// TIA Portal V20 export
DATA_BLOCK "InstCallEquipment"   // DB119
{ DB_Accessible_From_OPC_UA := 'FALSE' }
AUTHOR : ERsystem_FA2_DH. Kim
// stored: AssignedProDiagFB Unit1.Em5.ProDiag, DBAccessibleFromOPCUA false, DBAccessibleFromWebserver false, InstanceOfName Unit1.Em5.CallEquipment, InstanceOfType FB, Namespace Unit1.Em5
"Unit1.Em5.CallEquipment"
   // VAR_INPUT
   //    ZoneOperationEnable { ExternalWritable := 'False'} : "LWONIK_typeSafetyZoneManualOperation";
   // END_VAR
   // VAR_IN_OUT
   //    unitStatus : "LAF_typeUnitStatus";
   //    unitAlarmDB : "LAF_typeAlarms";
   //    emFeedback : "LUC_typeEmFeedback";
   // END_VAR
   // VAR
   //    InstSequenceMainPnP { S7_SetPoint := 'True'} : "Unit1.Em5.Sequence_1_MainPnP";
   //    InstSequenceAlignTable { S7_SetPoint := 'True'} : "Unit1.Em5.Sequence_2_AlignTable";
   //    InstSequenceNgPnP { S7_SetPoint := 'True'} : "Unit1.Em5.Sequence_3_NgPnP";
   //    InstSequenceGaugeRnR : "Unit1.Em5.Sequence_10_GaugeRnR";
   //    instMainPnPHomeJob10 : "LAF_SelectJob";
   //    instMainPnPHomeJob1 : "LAF_SelectJob";
   //    instMainPnPLoadJob2 : "LAF_SelectJob";
   //    instMainPnPUnloadJob3 : "LAF_SelectJob";
   //    instMainPnPAvoidJob4 : "LAF_SelectJob";
   //    instMainPnPOneLoadJob5 : "LAF_SelectJob";
   //    instMainPnPOneUnLoadJob6 : "LAF_SelectJob";
   //    instAlignTableHomeJob1 : "LAF_SelectJob";
   //    instAlignTableLoadJob2 : "LAF_SelectJob";
   //    instAlignTableVisionJob3 : "LAF_SelectJob";
   //    instAlignTableUnloadJob4 : "LAF_SelectJob";
   //    instAlignTableMotionJob22 : "LAF_SelectJob";
   //    instNgPnPHomeJob1 : "LAF_SelectJob";
   //    instNgPnPLoadJob2 : "LAF_SelectJob";
   //    instNgPnPUnloadJob3 : "LAF_SelectJob";
   //    instGaugeRnRCommonReadyJob1 : "LAF_SelectJob";
   //    instGaugeRnRCommonGetMasterPieceJob2 : "LAF_SelectJob";
   //    instGaugeRnRCommonMainPnPMoveAlignTableStackTableJob3 : "LAF_SelectJob";
   //    instGaugeRnRCommonMainPnp1ToAlignTableJob4 : "LAF_SelectJob";
   //    instGaugeRnRCommonMainPnPMoveReelCutConvyorAlignTableJob5 : "LAF_SelectJob";
   //    instGaugeRnRCommonAlignTableVisionAdjustJob6 : "LAF_SelectJob";
   //    instGaugeRnR1AlignAlignTableToMainPnP1Job10 { S7_SetPoint := 'True'} : "LAF_SelectJob";
   //    instGaugeRnR1AlignMainPnPMoveReelCutConvyorAlignTableJob11 { S7_SetPoint := 'True'} : "LAF_SelectJob";
   //    instGaugeRnR1AlignAlignTableMoveWaitJob12 { S7_SetPoint := 'True'} : "LAF_SelectJob";
   //    instGaugeRnR1AlignUnloadMasterPieceJob13 { S7_SetPoint := 'True'} : "LAF_SelectJob";
   //    instGaugeRnR1StackMainPnPMoveReelCutConvyorAlignTableJob15 { S7_SetPoint := 'True'} : "LAF_SelectJob";
   //    instGaugeRnR1StackAlignTableToMainPnP2Job16 { S7_SetPoint := 'True'} : "LAF_SelectJob";
   //    instGaugeRnR1StackMainPnPMoveAlignTableJob17 { S7_SetPoint := 'True'} : "LAF_SelectJob";
   //    instGaugeRnR1StackAlignTableMoveWaitJob18 { S7_SetPoint := 'True'} : "LAF_SelectJob";
   //    instGaugeRnR1StackMainPnP2ToStackTableJob19 { S7_SetPoint := 'True'} : "LAF_SelectJob";
   //    instGaugeRnR1StackStackTableToMainPnP2Job20 { S7_SetPoint := 'True'} : "LAF_SelectJob";
   //    instGaugeRnR1StackMainPnPMoveReelCutConvyorAlignTableJob21 { S7_SetPoint := 'True'} : "LAF_SelectJob";
   //    instGaugeRnR1StackMainPnP2ToAlignTableJob22 { S7_SetPoint := 'True'} : "LAF_SelectJob";
   //    instGaugeRnR1StackMainPnPMoveAlignTableJob23 { S7_SetPoint := 'True'} : "LAF_SelectJob";
   //    instGaugeRnR1StackAlignTableToMainPnP1Job24 { S7_SetPoint := 'True'} : "LAF_SelectJob";
   //    instGaugeRnR1StackMainPnPMoveReelCutConvyorAlignTableJob25 { S7_SetPoint := 'True'} : "LAF_SelectJob";
   //    instGaugeRnR1StackUnloadMasterPieceJob26 { S7_SetPoint := 'True'} : "LAF_SelectJob";
   //    instGaugeRnR3AlignMainPnPMoveReelCutConvyorAlignTableJob30 { S7_SetPoint := 'True'} : "LAF_SelectJob";
   //    instGaugeRnR3AlignNGPnPLoadMasterPieceJob31 { S7_SetPoint := 'True'} : "LAF_SelectJob";
   //    instGaugeRnR3AlignMainPnP2MoveAlignTableJob32 { S7_SetPoint := 'True'} : "LAF_SelectJob";
   //    instGaugeRnR3AlignAlignTableMoveWaitJob33 { S7_SetPoint := 'True'} : "LAF_SelectJob";
   //    instGaugeRnRCommonCheckCompleteJob39 { S7_SetPoint := 'True'} : "LAF_SelectJob";
   //    instCmPnp1stCathodeDetectSensor { S7_SetPoint := 'True'} : "LBC_DigitalSignalCn";
   //    instCmPnp2ndCathodeDetectSensor { S7_SetPoint := 'True'} : "LBC_DigitalSignalCn";
   //    instCmCathodeAlignTableElectrodeDetectSensor { S7_SetPoint := 'True'} : "LBC_DigitalSignalCn";
   //    instCmCathodeNgBoxFullSensorDetectSensor { S7_SetPoint := 'True'} : "LBC_DigitalSignalCn";
   //    instCmCathodeNgBoxDetectSensor { S7_SetPoint := 'True'} : "LBC_DigitalSignalCn";
   //    instCmCathodeMainPnP1AxisX { S7_SetPoint := 'True'} : "LBC_Axis64Pos_TecPlcCn";
   //    instCmCathodeMainPnP2AxisX { S7_SetPoint := 'True'} : "LBC_Axis64Pos_TecPlcCn";
   //    instCmCathodeMainPnP1AxisY { S7_SetPoint := 'True'} : "LBC_Axis64Pos_TecPlcCn";
   //    instCmCathodeMainPnP1AxisZ { S7_SetPoint := 'True'} : "LBC_Axis64Pos_TecPlcCn";
   //    instCmCathodeMainPnP2AxisZ { S7_SetPoint := 'True'} : "LBC_Axis64Pos_TecPlcCn";
   //    instCmCathodeAlignTableAxisX { S7_SetPoint := 'True'} : "LBC_Axis64Pos_TecPlcCn";
   //    instCmCathodeAlignTableAxisY1 { S7_SetPoint := 'True'} : "LBC_Axis64Pos_TecPlcCn";
   //    instCmCathodeAlignTableAxisY2 { S7_SetPoint := 'True'} : "LBC_Axis64Pos_TecPlcCn";
   //    instInterlockCathodeMainPnP1AxisX { S7_SetPoint := 'True'} : "LER_Axis64Pos_InterlockSummary";
   //    instInterlockCathodeMainPnP1AxisY { S7_SetPoint := 'True'} : "LER_Axis64Pos_InterlockSummary";
   //    instInterlockCathodeMainPnP1AxisZ { S7_SetPoint := 'True'} : "LER_Axis64Pos_InterlockSummary";
   //    instInterlockCathodeMainPnP2AxisX { S7_SetPoint := 'True'} : "LER_Axis64Pos_InterlockSummary";
   //    instInterlockCathodeMainPnP2AxisZ { S7_SetPoint := 'True'} : "LER_Axis64Pos_InterlockSummary";
   //    instInterlockCathodeAlignTableAxisX { S7_SetPoint := 'True'} : "LER_Axis64Pos_InterlockSummary";
   //    instInterlockCathodeAlignTableAxisY1 { S7_SetPoint := 'True'} : "LER_Axis64Pos_InterlockSummary";
   //    instInterlockCathodeAlignTableAxisY2 { S7_SetPoint := 'True'} : "LER_Axis64Pos_InterlockSummary";
   //    instCathodeMainPnP1AxisXSoftCam : "LER_SoftCam_Interface";
   //    instCathodeMainPnP2AxisXSoftCam { S7_SetPoint := 'True'} : "LER_SoftCam_Interface";
   //    instCathodeMainPnP1AxisYSoftCam { S7_SetPoint := 'True'} : "LER_SoftCam_Interface";
   //    instCathodeMainPnP1AxisZSoftCam { S7_SetPoint := 'True'} : "LER_SoftCam_Interface";
   //    instCathodeMainPnP2AxisZSoftCam { S7_SetPoint := 'True'} : "LER_SoftCam_Interface";
   //    instCathodeAlignTableAxisXSoftCam { S7_SetPoint := 'True'} : "LER_SoftCam_Interface";
   //    instCathodeAlignTableAxisY1SoftCam { S7_SetPoint := 'True'} : "LER_SoftCam_Interface";
   //    instCathodeAlignTableAxisY2SoftCam { S7_SetPoint := 'True'} : "LER_SoftCam_Interface";
   //    instCmCathodeMainPnP1RotaryCwCcw { ExternalAccessible := 'False'; ExternalVisible := 'False'; ExternalWritable := 'False'} : "LBC_TwoWayActuatorCn";
   //    instCmCathodeMainPnP1stSuctionPlateVacuum { ExternalAccessible := 'False'; ExternalVisible := 'False'; ExternalWritable := 'False'} : "LBC_TwoWayActuatorCn";
   //    instCmCathodeMainPnP2ndSuctionPlateVacuum { ExternalAccessible := 'False'; ExternalVisible := 'False'; ExternalWritable := 'False'} : "LBC_TwoWayActuatorCn";
   //    instCmCathodeAlignTableSuctionPlateVacuum { ExternalAccessible := 'False'; ExternalVisible := 'False'; ExternalWritable := 'False'; S7_SetPoint := 'True'} : "LBC_TwoWayActuatorCn";
   //    instCmCathodeGlassCleaning { ExternalAccessible := 'False'; ExternalVisible := 'False'; ExternalWritable := 'False'; S7_SetPoint := 'True'} : "LBC_TwoWayActuatorCn";
   //    instCmCathodeNgPnpUpDown { ExternalAccessible := 'False'; ExternalVisible := 'False'; ExternalWritable := 'False'; S7_SetPoint := 'True'} : "LBC_TwoWayActuatorCn";
   //    instCmCathodeNgPnp1stFwdBwd { ExternalAccessible := 'False'; ExternalVisible := 'False'; ExternalWritable := 'False'; S7_SetPoint := 'True'} : "LBC_TwoWayActuatorCn";
   //    instCmCathodeNgPnp2ndFwdBwd { ExternalAccessible := 'False'; ExternalVisible := 'False'; ExternalWritable := 'False'; S7_SetPoint := 'True'} : "LBC_TwoWayActuatorCn";
   //    instCmCathodeMaintenanceMovingFixFwdBwd { ExternalAccessible := 'False'; ExternalVisible := 'False'; ExternalWritable := 'False'; S7_SetPoint := 'True'} : "LBC_TwoWayActuatorCn";
   //    instCmCathodeNgBoxLiftUpDown { ExternalAccessible := 'False'; ExternalVisible := 'False'; ExternalWritable := 'False'; S7_SetPoint := 'True'} : "LBC_TwoWayActuatorCn";
   //    instCmCathodeNgBoxLockUpDown { ExternalAccessible := 'False'; ExternalVisible := 'False'; ExternalWritable := 'False'; S7_SetPoint := 'True'} : "LBC_TwoWayActuatorCn";
   //    instCmCathodeNgPnpVaccum { ExternalAccessible := 'False'; ExternalVisible := 'False'; ExternalWritable := 'False'; S7_SetPoint := 'True'} : "LBC_TwoWayActuatorCn";
   //    instCmCathodeConveyorCoverFwdBwd { S7_SetPoint := 'True'} : "LBC_TwoWayActuatorCn";
   //    instCmCathodeConveyorPickUpBlower { S7_SetPoint := 'True'} : "LBC_TwoWayActuatorCn";
   //    instCmCathodeVisionControllerInterface { ExternalAccessible := 'False'; ExternalVisible := 'False'; ExternalWritable := 'False'; S7_SetPoint := 'True'} : "LER_Vision_XGX2000";
   //    instAlignVisionConversion : "LER_AlignVisionConversion";
   //    instManageAlarms { ExternalWritable := 'False'} : "LAF_ManageAlarms";
   //    instEventsPFE : "Unit1.Em5.EventsPFE";
   //    instLER_BrakeTestCathodeMainPnP1AxisZ : "LER_BrakeTest";
   //    instLER_BrakeTestCathodeMainPnP2AxisZ { S7_SetPoint := 'True'} : "LER_BrakeTest";
   //    statUnitStatus { ExternalWritable := 'False'} : "LAF_typeUnitStatus";
   //    statSlmStatus : Struct
   //       running { ExternalWritable := 'False'} : Bool;
   //       powerOff { ExternalWritable := 'False'} : Bool;
   //    END_STRUCT;
   //    statAllBrakeTest { ExternalWritable := 'False'} : "LER_typeBrakeTestUnitCommands";
   //    statTonTime { ExternalAccessible := 'False'; ExternalVisible := 'False'; ExternalWritable := 'False'} : Array[0..1999] of TON_TIME;
   //    statTofTime { ExternalAccessible := 'False'; ExternalVisible := 'False'; ExternalWritable := 'False'} : Array[0..99] of TOF_TIME;
   //    statPulse { ExternalAccessible := 'False'; ExternalVisible := 'False'; ExternalWritable := 'False'} : Struct
   //       miscellaneous : Array[0..99] of Bool;
   //       workingDone : Struct
   //          mainPnP : Array[0..99] of Bool;
   //          alignTable : Array[0..99] of Bool;
   //          ngPnP : Array[0..99] of Bool;
   //       END_STRUCT;
   //       axisEnable : Array[0..99] of Bool;
   //       brakeTest : Array[0..99] of Bool;
   //    END_STRUCT;
   //    statEnableManualCmds : Bool := TRUE;
   //    Scan_on : Bool;
   //    "*** Interlock Axis ***" { ExternalAccessible := 'False'; ExternalVisible := 'False'; ExternalWritable := 'False'} : Bool;
   //    "cathodeMainPnP1AxisX Home" { S7_SetPoint := 'True'} : "Homing.LER_Axis";
   //    "cathodeMainPnP1AxisX Jog_CW" { S7_SetPoint := 'True'} : "Jog.LER_Axis";
   //    "cathodeMainPnP1AxisX Jog_CCW" { S7_SetPoint := 'True'} : "Jog.LER_Axis";
   //    "cathodeMainPnP1AxisX Position_" { S7_SetPoint := 'True'} : Array[0..5] of "Position.LER_Axis";
   //    "cathodeMainPnP2AxisX Home" { S7_SetPoint := 'True'} : "Homing.LER_Axis";
   //    "cathodeMainPnP2AxisX Jog_CW" { S7_SetPoint := 'True'} : "Jog.LER_Axis";
   //    "cathodeMainPnP2AxisX Jog_CCW" { S7_SetPoint := 'True'} : "Jog.LER_Axis";
   //    "cathodeMainPnP2AxisX Position_" { S7_SetPoint := 'True'} : Array[0..5] of "Position.LER_Axis";
   //    "cathodeMainPnP1AxisY Home" { S7_SetPoint := 'True'} : "Homing.LER_Axis";
   //    "cathodeMainPnP1AxisY Jog_CW" { S7_SetPoint := 'True'} : "Jog.LER_Axis";
   //    "cathodeMainPnP1AxisY Jog_CCW" { S7_SetPoint := 'True'} : "Jog.LER_Axis";
   //    "cathodeMainPnP1AxisY Position_" { S7_SetPoint := 'True'} : Array[0..5] of "Position.LER_Axis";
   //    "cathodeMainPnP1AxisZ Home" { S7_SetPoint := 'True'} : "Homing.LER_Axis";
   //    "cathodeMainPnP1AxisZ Jog_CW" { S7_SetPoint := 'True'} : "Jog.LER_Axis";
   //    "cathodeMainPnP1AxisZ Jog_CCW" { S7_SetPoint := 'True'} : "Jog.LER_Axis";
   //    "cathodeMainPnP1AxisZ Position_" { S7_SetPoint := 'True'} : Array[0..5] of "Position.LER_Axis";
   //    "cathodeMainPnP2AxisZ Home" { S7_SetPoint := 'True'} : "Homing.LER_Axis";
   //    "cathodeMainPnP2AxisZ Jog_CW" { S7_SetPoint := 'True'} : "Jog.LER_Axis";
   //    "cathodeMainPnP2AxisZ Jog_CCW" { S7_SetPoint := 'True'} : "Jog.LER_Axis";
   //    "cathodeMainPnP2AxisZ Position_" { S7_SetPoint := 'True'} : Array[0..5] of "Position.LER_Axis";
   //    "cathodeAlignTableAxisX Home" { S7_SetPoint := 'True'} : "Homing.LER_Axis";
   //    "cathodeAlignTableAxisX Jog_CW" { S7_SetPoint := 'True'} : "Jog.LER_Axis";
   //    "cathodeAlignTableAxisX Jog_CCW" { S7_SetPoint := 'True'} : "Jog.LER_Axis";
   //    "cathodeAlignTableAxisX Position_" { S7_SetPoint := 'True'} : Array[0..5] of "Position.LER_Axis";
   //    "cathodeAlignTableAxisY1 Home" { S7_SetPoint := 'True'} : "Homing.LER_Axis";
   //    "cathodeAlignTableAxisY1 Jog_CW" { S7_SetPoint := 'True'} : "Jog.LER_Axis";
   //    "cathodeAlignTableAxisY1 Jog_CCW" { S7_SetPoint := 'True'} : "Jog.LER_Axis";
   //    "cathodeAlignTableAxisY1 Position_" { S7_SetPoint := 'True'} : Array[0..5] of "Position.LER_Axis";
   //    "cathodeAlignTableAxisY2 Home" { S7_SetPoint := 'True'} : "Homing.LER_Axis";
   //    "cathodeAlignTableAxisY2 Jog_CW" { S7_SetPoint := 'True'} : "Jog.LER_Axis";
   //    "cathodeAlignTableAxisY2 Jog_CCW" { S7_SetPoint := 'True'} : "Jog.LER_Axis";
   //    "cathodeAlignTableAxisY2 Position_" { S7_SetPoint := 'True'} : Array[0..5] of "Position.LER_Axis";
   //    "*** Interlock Actuator ******" { ExternalAccessible := 'False'; ExternalVisible := 'False'; ExternalWritable := 'False'} : Bool;
   //    "cathodeNgBoxLiftUpDown Home" { S7_SetPoint := 'True'} : "Cylinder.LER_Actuator";
   //    "cathodeNgBoxLiftUpDown Work" { S7_SetPoint := 'True'} : "Cylinder.LER_Actuator";
   //    "cathodeNgBoxLockUpDown Home" { S7_SetPoint := 'True'} : "Cylinder.LER_Actuator";
   //    "cathodeNgBoxLockUpDown Work" { S7_SetPoint := 'True'} : "Cylinder.LER_Actuator";
   //    "cathodeMaintenanceMovingFixFrontFwdBwd Home" { S7_SetPoint := 'True'} : "Cylinder.LER_Actuator";
   //    "cathodeMaintenanceMovingFixFrontFwdBwd Work" { S7_SetPoint := 'True'} : "Cylinder.LER_Actuator";
   //    "cathodeGlassCleaning Home" { S7_SetPoint := 'True'} : "Cylinder.LER_Actuator";
   //    "cathodeGlassCleaning Work" { S7_SetPoint := 'True'} : "Cylinder.LER_Actuator";
   //    "cathodeNgPnp1stFwdBwd Home" { S7_SetPoint := 'True'} : "Cylinder.LER_Actuator";
   //    "cathodeNgPnp1stFwdBwd Work" { S7_SetPoint := 'True'} : "Cylinder.LER_Actuator";
   //    "cathodeNgPnpUpDown Home" { S7_SetPoint := 'True'} : "Cylinder.LER_Actuator";
   //    "cathodeNgPnpUpDown Work" { S7_SetPoint := 'True'} : "Cylinder.LER_Actuator";
   //    "cathodeMainPnP1RotaryCwCcw Home" { S7_SetPoint := 'True'} : "Cylinder.LER_Actuator";
   //    "cathodeMainPnP1RotaryCwCcw Work" { S7_SetPoint := 'True'} : "Cylinder.LER_Actuator";
   //    "cathodeNgPnp2ndFwdBwd Home" { S7_SetPoint := 'True'} : "Cylinder.LER_Actuator";
   //    "cathodeNgPnp2ndFwdBwd Work" { S7_SetPoint := 'True'} : "Cylinder.LER_Actuator";
   //    Tracking_05 { S7_SetPoint := 'True'} : "Unit1.Em5.PartData";
   //    AXIS7 : "LER_CM_Name";
   //    AXIS13 : "LER_CM_Name";
   //    AXIS18 : "LER_CM_Name";
   //    Cylinder23 : "LER_CM_Name";
   //    Cylinder28 : "LER_CM_Name";
   //    Vaccum15 : "LER_CM_Name";
   //    instAlignVisionHistory { S7_SetPoint := 'True'} : "LER_visionHistory";
   //    instAlignCalibration { S7_SetPoint := 'True'} : "LER_AlignCalibration";
   //    instAlignMoveCalibration { S7_SetPoint := 'True'} : "LER_AlignMoveCalibration";
   //    instAlignThetaCalibration { S7_SetPoint := 'True'} : "LER_AlignThetaCalibration";
   //    instAlignSyncMove { S7_SetPoint := 'True'} : "LER_AlignSyncMove";
   //    citi_Ptrig : Array[0..20] of Bool;
   //    citiTon : Array[0..20] of TON_TIME;
   //    citi : Time;
   //    citiTest : Array[0..20] of Bool;
   // END_VAR
BEGIN
   ZoneOperationEnable.autoStartEnable := FALSE;
   ZoneOperationEnable.doorLockEnable := TRUE;
   ZoneOperationEnable.doorUnlockEnable := TRUE;
   ZoneOperationEnable.rc_AutoEnable := FALSE;
   ZoneOperationEnable.rc_RollChangeEnable := FALSE;
   ZoneOperationEnable.rc_DoorLockEnable := TRUE;
   ZoneOperationEnable.rc_DoorUnlockEnable := TRUE;
   ZoneOperationEnable.hmiOperationEnable := TRUE;
   ZoneOperationEnable.phmiOperationEnable := FALSE;
   instCmPnp1stCathodeDetectSensor.enable := TRUE;
   instCmPnp1stCathodeDetectSensor.parentReferenceDesignator := WSTRING#'';
   instCmPnp1stCathodeDetectSensor.digitalValue := FALSE;
   instCmPnp1stCathodeDetectSensor.simulatedDigitalValue := FALSE;
   instCmPnp1stCathodeDetectSensor.statProcessValues.enable := TRUE;
   instCmPnp1stCathodeDetectSensor.statProcessValues.referenceDesignator := WSTRING#'DigitalSignal';
   instCmPnp1stCathodeDetectSensor.statProcessValues.simulation := FALSE;
   instCmPnp1stCathodeDetectSensor.statProcessValues.processValue := FALSE;
   instCmPnp1stCathodeDetectSensor.statProcessValues.error := FALSE;
   instCmPnp1stCathodeDetectSensor.statProcessValues.status := 16#0000;
   instCmPnp1stCathodeDetectSensor.statDiagnostics.status := 16#0000;
   instCmPnp1stCathodeDetectSensor.statDiagnostics.subfunctionStatus := 16#0000;
   instCmPnp1stCathodeDetectSensor.statDiagnostics.stateNumber := 0;
   instCmPnp1stCathodeDetectSensor.statEmptyDiagnostics.status := 16#0000;
   instCmPnp1stCathodeDetectSensor.statEmptyDiagnostics.subfunctionStatus := 16#0000;
   instCmPnp1stCathodeDetectSensor.statEmptyDiagnostics.stateNumber := 0;
   instCmPnp1stCathodeDetectSensor.instOnDelay.PT := T#0MS;
   instCmPnp1stCathodeDetectSensor.instOnDelay.IN := FALSE;
   instCmPnp1stCathodeDetectSensor.instOffDelay.PT := T#0MS;
   instCmPnp1stCathodeDetectSensor.instOffDelay.IN := FALSE;
   instCmPnp1stCathodeDetectSensor.statDisableAlarms := FALSE;
   instCmPnp1stCathodeDetectSensor.statErrorState := 16#0000;
   instCmPnp1stCathodeDetectSensor.statFirstCall := FALSE;
   instCmPnp1stCathodeDetectSensor.statResetPrevious := FALSE;
   instCmPnp1stCathodeDetectSensor.statEnablePrevious := TRUE;
   instCmPnp1stCathodeDetectSensor.statProcessValuePrevious := FALSE;
   instCmPnp2ndCathodeDetectSensor.enable := TRUE;
   instCmPnp2ndCathodeDetectSensor.parentReferenceDesignator := WSTRING#'';
   instCmPnp2ndCathodeDetectSensor.digitalValue := FALSE;
   instCmPnp2ndCathodeDetectSensor.simulatedDigitalValue := FALSE;
   instCmPnp2ndCathodeDetectSensor.statProcessValues.enable := TRUE;
   instCmPnp2ndCathodeDetectSensor.statProcessValues.referenceDesignator := WSTRING#'DigitalSignal';
   instCmPnp2ndCathodeDetectSensor.statProcessValues.simulation := FALSE;
   instCmPnp2ndCathodeDetectSensor.statProcessValues.processValue := FALSE;
   instCmPnp2ndCathodeDetectSensor.statProcessValues.error := FALSE;
   instCmPnp2ndCathodeDetectSensor.statProcessValues.status := 16#0000;
   instCmPnp2ndCathodeDetectSensor.statDiagnostics.status := 16#0000;
   instCmPnp2ndCathodeDetectSensor.statDiagnostics.subfunctionStatus := 16#0000;
   instCmPnp2ndCathodeDetectSensor.statDiagnostics.stateNumber := 0;
   instCmPnp2ndCathodeDetectSensor.statEmptyDiagnostics.status := 16#0000;
   instCmPnp2ndCathodeDetectSensor.statEmptyDiagnostics.subfunctionStatus := 16#0000;
   instCmPnp2ndCathodeDetectSensor.statEmptyDiagnostics.stateNumber := 0;
   instCmPnp2ndCathodeDetectSensor.instOnDelay.PT := T#0MS;
   instCmPnp2ndCathodeDetectSensor.instOnDelay.IN := FALSE;
   instCmPnp2ndCathodeDetectSensor.instOffDelay.PT := T#0MS;
   instCmPnp2ndCathodeDetectSensor.instOffDelay.IN := FALSE;
   instCmPnp2ndCathodeDetectSensor.statDisableAlarms := FALSE;
   instCmPnp2ndCathodeDetectSensor.statErrorState := 16#0000;
   instCmPnp2ndCathodeDetectSensor.statFirstCall := FALSE;
   instCmPnp2ndCathodeDetectSensor.statResetPrevious := FALSE;
   instCmPnp2ndCathodeDetectSensor.statEnablePrevious := TRUE;
   instCmPnp2ndCathodeDetectSensor.statProcessValuePrevious := FALSE;
   instCmCathodeAlignTableElectrodeDetectSensor.enable := TRUE;
   instCmCathodeAlignTableElectrodeDetectSensor.parentReferenceDesignator := WSTRING#'';
   instCmCathodeAlignTableElectrodeDetectSensor.digitalValue := FALSE;
   instCmCathodeAlignTableElectrodeDetectSensor.simulatedDigitalValue := FALSE;
   instCmCathodeAlignTableElectrodeDetectSensor.statProcessValues.enable := TRUE;
   instCmCathodeAlignTableElectrodeDetectSensor.statProcessValues.referenceDesignator := WSTRING#'DigitalSignal';
   instCmCathodeAlignTableElectrodeDetectSensor.statProcessValues.simulation := FALSE;
   instCmCathodeAlignTableElectrodeDetectSensor.statProcessValues.processValue := FALSE;
   instCmCathodeAlignTableElectrodeDetectSensor.statProcessValues.error := FALSE;
   instCmCathodeAlignTableElectrodeDetectSensor.statProcessValues.status := 16#0000;
   instCmCathodeAlignTableElectrodeDetectSensor.statDiagnostics.status := 16#0000;
   instCmCathodeAlignTableElectrodeDetectSensor.statDiagnostics.subfunctionStatus := 16#0000;
   instCmCathodeAlignTableElectrodeDetectSensor.statDiagnostics.stateNumber := 0;
   instCmCathodeAlignTableElectrodeDetectSensor.statEmptyDiagnostics.status := 16#0000;
   instCmCathodeAlignTableElectrodeDetectSensor.statEmptyDiagnostics.subfunctionStatus := 16#0000;
   instCmCathodeAlignTableElectrodeDetectSensor.statEmptyDiagnostics.stateNumber := 0;
   instCmCathodeAlignTableElectrodeDetectSensor.instOnDelay.PT := T#0MS;
   instCmCathodeAlignTableElectrodeDetectSensor.instOnDelay.IN := FALSE;
   instCmCathodeAlignTableElectrodeDetectSensor.instOffDelay.PT := T#0MS;
   instCmCathodeAlignTableElectrodeDetectSensor.instOffDelay.IN := FALSE;
   instCmCathodeAlignTableElectrodeDetectSensor.statDisableAlarms := FALSE;
   instCmCathodeAlignTableElectrodeDetectSensor.statErrorState := 16#0000;
   instCmCathodeAlignTableElectrodeDetectSensor.statFirstCall := FALSE;
   instCmCathodeAlignTableElectrodeDetectSensor.statResetPrevious := FALSE;
   instCmCathodeAlignTableElectrodeDetectSensor.statEnablePrevious := TRUE;
   instCmCathodeAlignTableElectrodeDetectSensor.statProcessValuePrevious := FALSE;
   instCmCathodeNgBoxFullSensorDetectSensor.enable := TRUE;
   instCmCathodeNgBoxFullSensorDetectSensor.parentReferenceDesignator := WSTRING#'';
   instCmCathodeNgBoxFullSensorDetectSensor.digitalValue := FALSE;
   instCmCathodeNgBoxFullSensorDetectSensor.simulatedDigitalValue := FALSE;
   instCmCathodeNgBoxFullSensorDetectSensor.statProcessValues.enable := TRUE;
   instCmCathodeNgBoxFullSensorDetectSensor.statProcessValues.referenceDesignator := WSTRING#'DigitalSignal';
   instCmCathodeNgBoxFullSensorDetectSensor.statProcessValues.simulation := FALSE;
   instCmCathodeNgBoxFullSensorDetectSensor.statProcessValues.processValue := FALSE;
   instCmCathodeNgBoxFullSensorDetectSensor.statProcessValues.error := FALSE;
   instCmCathodeNgBoxFullSensorDetectSensor.statProcessValues.status := 16#0000;
   instCmCathodeNgBoxFullSensorDetectSensor.statDiagnostics.status := 16#0000;
   instCmCathodeNgBoxFullSensorDetectSensor.statDiagnostics.subfunctionStatus := 16#0000;
   instCmCathodeNgBoxFullSensorDetectSensor.statDiagnostics.stateNumber := 0;
   instCmCathodeNgBoxFullSensorDetectSensor.statEmptyDiagnostics.status := 16#0000;
   instCmCathodeNgBoxFullSensorDetectSensor.statEmptyDiagnostics.subfunctionStatus := 16#0000;
   instCmCathodeNgBoxFullSensorDetectSensor.statEmptyDiagnostics.stateNumber := 0;
   instCmCathodeNgBoxFullSensorDetectSensor.instOnDelay.PT := T#0MS;
   instCmCathodeNgBoxFullSensorDetectSensor.instOnDelay.IN := FALSE;
   instCmCathodeNgBoxFullSensorDetectSensor.instOffDelay.PT := T#0MS;
   instCmCathodeNgBoxFullSensorDetectSensor.instOffDelay.IN := FALSE;
   instCmCathodeNgBoxFullSensorDetectSensor.statDisableAlarms := FALSE;
   instCmCathodeNgBoxFullSensorDetectSensor.statErrorState := 16#0000;
   instCmCathodeNgBoxFullSensorDetectSensor.statFirstCall := FALSE;
   instCmCathodeNgBoxFullSensorDetectSensor.statResetPrevious := FALSE;
   instCmCathodeNgBoxFullSensorDetectSensor.statEnablePrevious := TRUE;
   instCmCathodeNgBoxFullSensorDetectSensor.statProcessValuePrevious := FALSE;
   instCmCathodeNgBoxDetectSensor.enable := TRUE;
   instCmCathodeNgBoxDetectSensor.parentReferenceDesignator := WSTRING#'';
   instCmCathodeNgBoxDetectSensor.digitalValue := TRUE;
   instCmCathodeNgBoxDetectSensor.simulatedDigitalValue := FALSE;
   instCmCathodeNgBoxDetectSensor.statProcessValues.enable := TRUE;
   instCmCathodeNgBoxDetectSensor.statProcessValues.referenceDesignator := WSTRING#'DigitalSignal';
   instCmCathodeNgBoxDetectSensor.statProcessValues.simulation := FALSE;
   instCmCathodeNgBoxDetectSensor.statProcessValues.processValue := TRUE;
   instCmCathodeNgBoxDetectSensor.statProcessValues.error := FALSE;
   instCmCathodeNgBoxDetectSensor.statProcessValues.status := 16#0000;
   instCmCathodeNgBoxDetectSensor.statDiagnostics.status := 16#0000;
   instCmCathodeNgBoxDetectSensor.statDiagnostics.subfunctionStatus := 16#0000;
   instCmCathodeNgBoxDetectSensor.statDiagnostics.stateNumber := 0;
   instCmCathodeNgBoxDetectSensor.statEmptyDiagnostics.status := 16#0000;
   instCmCathodeNgBoxDetectSensor.statEmptyDiagnostics.subfunctionStatus := 16#0000;
   instCmCathodeNgBoxDetectSensor.statEmptyDiagnostics.stateNumber := 0;
   instCmCathodeNgBoxDetectSensor.instOnDelay.PT := T#0MS;
   instCmCathodeNgBoxDetectSensor.instOnDelay.IN := FALSE;
   instCmCathodeNgBoxDetectSensor.instOffDelay.PT := T#0MS;
   instCmCathodeNgBoxDetectSensor.instOffDelay.IN := FALSE;
   instCmCathodeNgBoxDetectSensor.statDisableAlarms := FALSE;
   instCmCathodeNgBoxDetectSensor.statErrorState := 16#0000;
   instCmCathodeNgBoxDetectSensor.statFirstCall := FALSE;
   instCmCathodeNgBoxDetectSensor.statResetPrevious := FALSE;
   instCmCathodeNgBoxDetectSensor.statEnablePrevious := TRUE;
   instCmCathodeNgBoxDetectSensor.statProcessValuePrevious := TRUE;
   instCmCathodeMainPnP1RotaryCwCcw.enable := TRUE;
   instCmCathodeMainPnP1RotaryCwCcw.parentReferenceDesignator := WSTRING#'';
   instCmCathodeMainPnP1RotaryCwCcw.feedbackHomePos := FALSE;
   instCmCathodeMainPnP1RotaryCwCcw.feedbackWorkPos := TRUE;
   instCmCathodeMainPnP1RotaryCwCcw.enableManualCmds := TRUE;
   instCmCathodeMainPnP1RotaryCwCcw.interlockWorkPos := FALSE;
   instCmCathodeMainPnP1RotaryCwCcw.interlockHomePos := FALSE;
   instCmCathodeMainPnP1RotaryCwCcw.goToHomePos := FALSE;
   instCmCathodeMainPnP1RotaryCwCcw.goToWorkPos := FALSE;
   instCmCathodeMainPnP1RotaryCwCcw.statProcessValues.enable := TRUE;
   instCmCathodeMainPnP1RotaryCwCcw.statProcessValues.referenceDesignator := WSTRING#'MainPnP1RotaryCwCcw';
   instCmCathodeMainPnP1RotaryCwCcw.statProcessValues.commandHomePos := FALSE;
   instCmCathodeMainPnP1RotaryCwCcw.statProcessValues.commandWorkPos := FALSE;
   instCmCathodeMainPnP1RotaryCwCcw.statProcessValues.goToHomePos := FALSE;
   instCmCathodeMainPnP1RotaryCwCcw.statProcessValues.goToWorkPos := FALSE;
   instCmCathodeMainPnP1RotaryCwCcw.statProcessValues.inHomePos := FALSE;
   instCmCathodeMainPnP1RotaryCwCcw.statProcessValues.inWorkPos := TRUE;
   instCmCathodeMainPnP1RotaryCwCcw.statProcessValues.reset := FALSE;
   instCmCathodeMainPnP1RotaryCwCcw.statProcessValues.enableManualCmds := TRUE;
   instCmCathodeMainPnP1RotaryCwCcw.statProcessValues.error := FALSE;
   instCmCathodeMainPnP1RotaryCwCcw.statProcessValues.interlockHomePos := FALSE;
   instCmCathodeMainPnP1RotaryCwCcw.statProcessValues.interlockWorkPos := FALSE;
   instCmCathodeMainPnP1RotaryCwCcw.statProcessValues.status := 16#7100;
   instCmCathodeMainPnP1RotaryCwCcw.statProcessValues.interlockWarningWorkPos := FALSE;
   instCmCathodeMainPnP1RotaryCwCcw.statProcessValues.interlockWarningHomePos := FALSE;
   instCmCathodeMainPnP1RotaryCwCcw.statCurrentInputs.commandHomePos := FALSE;
   instCmCathodeMainPnP1RotaryCwCcw.statCurrentInputs.commandWorkPos := FALSE;
   instCmCathodeMainPnP1RotaryCwCcw.statCurrentInputs.reset := FALSE;
   instCmCathodeMainPnP1RotaryCwCcw.statPreviousInputs.commandHomePos := FALSE;
   instCmCathodeMainPnP1RotaryCwCcw.statPreviousInputs.commandWorkPos := FALSE;
   instCmCathodeMainPnP1RotaryCwCcw.statPreviousInputs.reset := FALSE;
   instCmCathodeMainPnP1RotaryCwCcw.statCurrentInterface.commandHomePos := FALSE;
   instCmCathodeMainPnP1RotaryCwCcw.statCurrentInterface.commandWorkPos := FALSE;
   instCmCathodeMainPnP1RotaryCwCcw.statCurrentInterface.reset := FALSE;
   instCmCathodeMainPnP1RotaryCwCcw.statPreviousInterface.commandHomePos := FALSE;
   instCmCathodeMainPnP1RotaryCwCcw.statPreviousInterface.commandWorkPos := FALSE;
   instCmCathodeMainPnP1RotaryCwCcw.statPreviousInterface.reset := FALSE;
   instCmCathodeMainPnP1RotaryCwCcw.statEmptyDiagnostics.status := 16#0000;
   instCmCathodeMainPnP1RotaryCwCcw.statEmptyDiagnostics.subfunctionStatus := 16#0000;
   instCmCathodeMainPnP1RotaryCwCcw.statEmptyDiagnostics.stateNumber := 0;
   instCmCathodeMainPnP1RotaryCwCcw.instTimerReachPos.PT := T#0MS;
   instCmCathodeMainPnP1RotaryCwCcw.instTimerReachPos.IN := FALSE;
   instCmCathodeMainPnP1RotaryCwCcw.instTimerLeavePos.PT := T#0MS;
   instCmCathodeMainPnP1RotaryCwCcw.instTimerLeavePos.IN := FALSE;
   instCmCathodeMainPnP1RotaryCwCcw.instTimerDiscrepancyCheck.PT := T#0MS;
   instCmCathodeMainPnP1RotaryCwCcw.instTimerDiscrepancyCheck.IN := FALSE;
   instCmCathodeMainPnP1RotaryCwCcw.statDisableAlarms := TRUE;
   instCmCathodeMainPnP1RotaryCwCcw.statDiagnostics.status := 16#7003;
   instCmCathodeMainPnP1RotaryCwCcw.statDiagnostics.subfunctionStatus := 16#0000;
   instCmCathodeMainPnP1RotaryCwCcw.statDiagnostics.stateNumber := 0;
   instCmCathodeMainPnP1RotaryCwCcw.statEnablePrevious := TRUE;
   instCmCathodeMainPnP1RotaryCwCcw.statFirstCall := FALSE;
   instCmCathodeMainPnP1RotaryCwCcw.statResetPrevious := FALSE;
   instCmCathodeMainPnP1RotaryCwCcw.statValid := TRUE;
   instCmCathodeMainPnP1RotaryCwCcw.statBusy := TRUE;
   instCmCathodeMainPnP1RotaryCwCcw.statError := FALSE;
   instCmCathodeMainPnP1RotaryCwCcw.statInterlockWorkOff := FALSE;
   instCmCathodeMainPnP1RotaryCwCcw.statInterlockHomeOff := FALSE;
   instCmCathodeMainPnP1RotaryCwCcw.statFbState := 50;
   instCmCathodeMainPnP1RotaryCwCcw.statFbStatePrevious := 50;
   instCmCathodeMainPnP1RotaryCwCcw.statErrorUserCleared := FALSE;
   instCmCathodeMainPnP1RotaryCwCcw.statErrorAutoCleared := FALSE;
   instCmCathodeMainPnP1RotaryCwCcw.statErrorState := 16#0000;
   instCmCathodeMainPnP1RotaryCwCcw.statDisablingCompleted := FALSE;
   instCmCathodeMainPnP1RotaryCwCcw.statFeedbackHomePos := FALSE;
   instCmCathodeMainPnP1RotaryCwCcw.statFeedbackWorkPos := TRUE;
   instCmCathodeMainPnP1stSuctionPlateVacuum.enable := TRUE;
   instCmCathodeMainPnP1stSuctionPlateVacuum.parentReferenceDesignator := WSTRING#'';
   instCmCathodeMainPnP1stSuctionPlateVacuum.feedbackHomePos := TRUE;
   instCmCathodeMainPnP1stSuctionPlateVacuum.feedbackWorkPos := FALSE;
   instCmCathodeMainPnP1stSuctionPlateVacuum.enableManualCmds := TRUE;
   instCmCathodeMainPnP1stSuctionPlateVacuum.interlockWorkPos := TRUE;
   instCmCathodeMainPnP1stSuctionPlateVacuum.interlockHomePos := TRUE;
   instCmCathodeMainPnP1stSuctionPlateVacuum.goToHomePos := FALSE;
   instCmCathodeMainPnP1stSuctionPlateVacuum.goToWorkPos := FALSE;
   instCmCathodeMainPnP1stSuctionPlateVacuum.statProcessValues.enable := TRUE;
   instCmCathodeMainPnP1stSuctionPlateVacuum.statProcessValues.referenceDesignator := WSTRING#'MainPnP1Vacuum';
   instCmCathodeMainPnP1stSuctionPlateVacuum.statProcessValues.commandHomePos := FALSE;
   instCmCathodeMainPnP1stSuctionPlateVacuum.statProcessValues.commandWorkPos := FALSE;
   instCmCathodeMainPnP1stSuctionPlateVacuum.statProcessValues.goToHomePos := FALSE;
   instCmCathodeMainPnP1stSuctionPlateVacuum.statProcessValues.goToWorkPos := FALSE;
   instCmCathodeMainPnP1stSuctionPlateVacuum.statProcessValues.inHomePos := TRUE;
   instCmCathodeMainPnP1stSuctionPlateVacuum.statProcessValues.inWorkPos := FALSE;
   instCmCathodeMainPnP1stSuctionPlateVacuum.statProcessValues.reset := FALSE;
   instCmCathodeMainPnP1stSuctionPlateVacuum.statProcessValues.enableManualCmds := TRUE;
   instCmCathodeMainPnP1stSuctionPlateVacuum.statProcessValues.error := FALSE;
   instCmCathodeMainPnP1stSuctionPlateVacuum.statProcessValues.interlockHomePos := TRUE;
   instCmCathodeMainPnP1stSuctionPlateVacuum.statProcessValues.interlockWorkPos := TRUE;
   instCmCathodeMainPnP1stSuctionPlateVacuum.statProcessValues.status := 16#7003;
   instCmCathodeMainPnP1stSuctionPlateVacuum.statProcessValues.interlockWarningWorkPos := FALSE;
   instCmCathodeMainPnP1stSuctionPlateVacuum.statProcessValues.interlockWarningHomePos := FALSE;
   instCmCathodeMainPnP1stSuctionPlateVacuum.statCurrentInputs.commandHomePos := FALSE;
   instCmCathodeMainPnP1stSuctionPlateVacuum.statCurrentInputs.commandWorkPos := FALSE;
   instCmCathodeMainPnP1stSuctionPlateVacuum.statCurrentInputs.reset := FALSE;
   instCmCathodeMainPnP1stSuctionPlateVacuum.statPreviousInputs.commandHomePos := FALSE;
   instCmCathodeMainPnP1stSuctionPlateVacuum.statPreviousInputs.commandWorkPos := FALSE;
   instCmCathodeMainPnP1stSuctionPlateVacuum.statPreviousInputs.reset := FALSE;
   instCmCathodeMainPnP1stSuctionPlateVacuum.statCurrentInterface.commandHomePos := FALSE;
   instCmCathodeMainPnP1stSuctionPlateVacuum.statCurrentInterface.commandWorkPos := FALSE;
   instCmCathodeMainPnP1stSuctionPlateVacuum.statCurrentInterface.reset := FALSE;
   instCmCathodeMainPnP1stSuctionPlateVacuum.statPreviousInterface.commandHomePos := FALSE;
   instCmCathodeMainPnP1stSuctionPlateVacuum.statPreviousInterface.commandWorkPos := FALSE;
   instCmCathodeMainPnP1stSuctionPlateVacuum.statPreviousInterface.reset := FALSE;
   instCmCathodeMainPnP1stSuctionPlateVacuum.statEmptyDiagnostics.status := 16#0000;
   instCmCathodeMainPnP1stSuctionPlateVacuum.statEmptyDiagnostics.subfunctionStatus := 16#0000;
   instCmCathodeMainPnP1stSuctionPlateVacuum.statEmptyDiagnostics.stateNumber := 0;
   instCmCathodeMainPnP1stSuctionPlateVacuum.instTimerReachPos.PT := T#0MS;
   instCmCathodeMainPnP1stSuctionPlateVacuum.instTimerReachPos.IN := FALSE;
   instCmCathodeMainPnP1stSuctionPlateVacuum.instTimerLeavePos.PT := T#0MS;
   instCmCathodeMainPnP1stSuctionPlateVacuum.instTimerLeavePos.IN := FALSE;
   instCmCathodeMainPnP1stSuctionPlateVacuum.instTimerDiscrepancyCheck.PT := T#0MS;
   instCmCathodeMainPnP1stSuctionPlateVacuum.instTimerDiscrepancyCheck.IN := FALSE;
   instCmCathodeMainPnP1stSuctionPlateVacuum.statDisableAlarms := FALSE;
   instCmCathodeMainPnP1stSuctionPlateVacuum.statDiagnostics.status := 16#7003;
   instCmCathodeMainPnP1stSuctionPlateVacuum.statDiagnostics.subfunctionStatus := 16#0000;
   instCmCathodeMainPnP1stSuctionPlateVacuum.statDiagnostics.stateNumber := 0;
   instCmCathodeMainPnP1stSuctionPlateVacuum.statEnablePrevious := TRUE;
   instCmCathodeMainPnP1stSuctionPlateVacuum.statFirstCall := FALSE;
   instCmCathodeMainPnP1stSuctionPlateVacuum.statResetPrevious := FALSE;
   instCmCathodeMainPnP1stSuctionPlateVacuum.statValid := TRUE;
   instCmCathodeMainPnP1stSuctionPlateVacuum.statBusy := TRUE;
   instCmCathodeMainPnP1stSuctionPlateVacuum.statError := FALSE;
   instCmCathodeMainPnP1stSuctionPlateVacuum.statInterlockWorkOff := FALSE;
   instCmCathodeMainPnP1stSuctionPlateVacuum.statInterlockHomeOff := FALSE;
   instCmCathodeMainPnP1stSuctionPlateVacuum.statFbState := 50;
   instCmCathodeMainPnP1stSuctionPlateVacuum.statFbStatePrevious := 50;
   instCmCathodeMainPnP1stSuctionPlateVacuum.statErrorUserCleared := FALSE;
   instCmCathodeMainPnP1stSuctionPlateVacuum.statErrorAutoCleared := FALSE;
   instCmCathodeMainPnP1stSuctionPlateVacuum.statErrorState := 16#0000;
   instCmCathodeMainPnP1stSuctionPlateVacuum.statDisablingCompleted := FALSE;
   instCmCathodeMainPnP1stSuctionPlateVacuum.statFeedbackHomePos := TRUE;
   instCmCathodeMainPnP1stSuctionPlateVacuum.statFeedbackWorkPos := FALSE;
   instCmCathodeMainPnP2ndSuctionPlateVacuum.enable := TRUE;
   instCmCathodeMainPnP2ndSuctionPlateVacuum.parentReferenceDesignator := WSTRING#'';
   instCmCathodeMainPnP2ndSuctionPlateVacuum.feedbackHomePos := TRUE;
   instCmCathodeMainPnP2ndSuctionPlateVacuum.feedbackWorkPos := FALSE;
   instCmCathodeMainPnP2ndSuctionPlateVacuum.enableManualCmds := TRUE;
   instCmCathodeMainPnP2ndSuctionPlateVacuum.interlockWorkPos := TRUE;
   instCmCathodeMainPnP2ndSuctionPlateVacuum.interlockHomePos := TRUE;
   instCmCathodeMainPnP2ndSuctionPlateVacuum.goToHomePos := FALSE;
   instCmCathodeMainPnP2ndSuctionPlateVacuum.goToWorkPos := FALSE;
   instCmCathodeMainPnP2ndSuctionPlateVacuum.statProcessValues.enable := TRUE;
   instCmCathodeMainPnP2ndSuctionPlateVacuum.statProcessValues.referenceDesignator := WSTRING#'MainPnP2Vacuum';
   instCmCathodeMainPnP2ndSuctionPlateVacuum.statProcessValues.commandHomePos := FALSE;
   instCmCathodeMainPnP2ndSuctionPlateVacuum.statProcessValues.commandWorkPos := FALSE;
   instCmCathodeMainPnP2ndSuctionPlateVacuum.statProcessValues.goToHomePos := FALSE;
   instCmCathodeMainPnP2ndSuctionPlateVacuum.statProcessValues.goToWorkPos := FALSE;
   instCmCathodeMainPnP2ndSuctionPlateVacuum.statProcessValues.inHomePos := TRUE;
   instCmCathodeMainPnP2ndSuctionPlateVacuum.statProcessValues.inWorkPos := FALSE;
   instCmCathodeMainPnP2ndSuctionPlateVacuum.statProcessValues.reset := FALSE;
   instCmCathodeMainPnP2ndSuctionPlateVacuum.statProcessValues.enableManualCmds := TRUE;
   instCmCathodeMainPnP2ndSuctionPlateVacuum.statProcessValues.error := FALSE;
   instCmCathodeMainPnP2ndSuctionPlateVacuum.statProcessValues.interlockHomePos := TRUE;
   instCmCathodeMainPnP2ndSuctionPlateVacuum.statProcessValues.interlockWorkPos := TRUE;
   instCmCathodeMainPnP2ndSuctionPlateVacuum.statProcessValues.status := 16#7003;
   instCmCathodeMainPnP2ndSuctionPlateVacuum.statProcessValues.interlockWarningWorkPos := FALSE;
   instCmCathodeMainPnP2ndSuctionPlateVacuum.statProcessValues.interlockWarningHomePos := FALSE;
   instCmCathodeMainPnP2ndSuctionPlateVacuum.statCurrentInputs.commandHomePos := FALSE;
   instCmCathodeMainPnP2ndSuctionPlateVacuum.statCurrentInputs.commandWorkPos := FALSE;
   instCmCathodeMainPnP2ndSuctionPlateVacuum.statCurrentInputs.reset := FALSE;
   instCmCathodeMainPnP2ndSuctionPlateVacuum.statPreviousInputs.commandHomePos := FALSE;
   instCmCathodeMainPnP2ndSuctionPlateVacuum.statPreviousInputs.commandWorkPos := FALSE;
   instCmCathodeMainPnP2ndSuctionPlateVacuum.statPreviousInputs.reset := FALSE;
   instCmCathodeMainPnP2ndSuctionPlateVacuum.statCurrentInterface.commandHomePos := FALSE;
   instCmCathodeMainPnP2ndSuctionPlateVacuum.statCurrentInterface.commandWorkPos := FALSE;
   instCmCathodeMainPnP2ndSuctionPlateVacuum.statCurrentInterface.reset := FALSE;
   instCmCathodeMainPnP2ndSuctionPlateVacuum.statPreviousInterface.commandHomePos := FALSE;
   instCmCathodeMainPnP2ndSuctionPlateVacuum.statPreviousInterface.commandWorkPos := FALSE;
   instCmCathodeMainPnP2ndSuctionPlateVacuum.statPreviousInterface.reset := FALSE;
   instCmCathodeMainPnP2ndSuctionPlateVacuum.statEmptyDiagnostics.status := 16#0000;
   instCmCathodeMainPnP2ndSuctionPlateVacuum.statEmptyDiagnostics.subfunctionStatus := 16#0000;
   instCmCathodeMainPnP2ndSuctionPlateVacuum.statEmptyDiagnostics.stateNumber := 0;
   instCmCathodeMainPnP2ndSuctionPlateVacuum.instTimerReachPos.PT := T#0MS;
   instCmCathodeMainPnP2ndSuctionPlateVacuum.instTimerReachPos.IN := FALSE;
   instCmCathodeMainPnP2ndSuctionPlateVacuum.instTimerLeavePos.PT := T#0MS;
   instCmCathodeMainPnP2ndSuctionPlateVacuum.instTimerLeavePos.IN := FALSE;
   instCmCathodeMainPnP2ndSuctionPlateVacuum.instTimerDiscrepancyCheck.PT := T#0MS;
   instCmCathodeMainPnP2ndSuctionPlateVacuum.instTimerDiscrepancyCheck.IN := FALSE;
   instCmCathodeMainPnP2ndSuctionPlateVacuum.statDisableAlarms := FALSE;
   instCmCathodeMainPnP2ndSuctionPlateVacuum.statDiagnostics.status := 16#7003;
   instCmCathodeMainPnP2ndSuctionPlateVacuum.statDiagnostics.subfunctionStatus := 16#0000;
   instCmCathodeMainPnP2ndSuctionPlateVacuum.statDiagnostics.stateNumber := 0;
   instCmCathodeMainPnP2ndSuctionPlateVacuum.statEnablePrevious := TRUE;
   instCmCathodeMainPnP2ndSuctionPlateVacuum.statFirstCall := FALSE;
   instCmCathodeMainPnP2ndSuctionPlateVacuum.statResetPrevious := FALSE;
   instCmCathodeMainPnP2ndSuctionPlateVacuum.statValid := TRUE;
   instCmCathodeMainPnP2ndSuctionPlateVacuum.statBusy := TRUE;
   instCmCathodeMainPnP2ndSuctionPlateVacuum.statError := FALSE;
   instCmCathodeMainPnP2ndSuctionPlateVacuum.statInterlockWorkOff := FALSE;
   instCmCathodeMainPnP2ndSuctionPlateVacuum.statInterlockHomeOff := FALSE;
   instCmCathodeMainPnP2ndSuctionPlateVacuum.statFbState := 50;
   instCmCathodeMainPnP2ndSuctionPlateVacuum.statFbStatePrevious := 50;
   instCmCathodeMainPnP2ndSuctionPlateVacuum.statErrorUserCleared := FALSE;
   instCmCathodeMainPnP2ndSuctionPlateVacuum.statErrorAutoCleared := FALSE;
   instCmCathodeMainPnP2ndSuctionPlateVacuum.statErrorState := 16#0000;
   instCmCathodeMainPnP2ndSuctionPlateVacuum.statDisablingCompleted := FALSE;
   instCmCathodeMainPnP2ndSuctionPlateVacuum.statFeedbackHomePos := TRUE;
   instCmCathodeMainPnP2ndSuctionPlateVacuum.statFeedbackWorkPos := FALSE;
   instCmCathodeAlignTableSuctionPlateVacuum.enable := TRUE;
   instCmCathodeAlignTableSuctionPlateVacuum.parentReferenceDesignator := WSTRING#'';
   instCmCathodeAlignTableSuctionPlateVacuum.feedbackHomePos := TRUE;
   instCmCathodeAlignTableSuctionPlateVacuum.feedbackWorkPos := FALSE;
   instCmCathodeAlignTableSuctionPlateVacuum.enableManualCmds := TRUE;
   instCmCathodeAlignTableSuctionPlateVacuum.interlockWorkPos := TRUE;
   instCmCathodeAlignTableSuctionPlateVacuum.interlockHomePos := TRUE;
   instCmCathodeAlignTableSuctionPlateVacuum.goToHomePos := FALSE;
   instCmCathodeAlignTableSuctionPlateVacuum.goToWorkPos := FALSE;
   instCmCathodeAlignTableSuctionPlateVacuum.statProcessValues.enable := TRUE;
   instCmCathodeAlignTableSuctionPlateVacuum.statProcessValues.referenceDesignator := WSTRING#'AlignTableVaccum';
   instCmCathodeAlignTableSuctionPlateVacuum.statProcessValues.commandHomePos := FALSE;
   instCmCathodeAlignTableSuctionPlateVacuum.statProcessValues.commandWorkPos := FALSE;
   instCmCathodeAlignTableSuctionPlateVacuum.statProcessValues.goToHomePos := FALSE;
   instCmCathodeAlignTableSuctionPlateVacuum.statProcessValues.goToWorkPos := FALSE;
   instCmCathodeAlignTableSuctionPlateVacuum.statProcessValues.inHomePos := TRUE;
   instCmCathodeAlignTableSuctionPlateVacuum.statProcessValues.inWorkPos := FALSE;
   instCmCathodeAlignTableSuctionPlateVacuum.statProcessValues.reset := FALSE;
   instCmCathodeAlignTableSuctionPlateVacuum.statProcessValues.enableManualCmds := TRUE;
   instCmCathodeAlignTableSuctionPlateVacuum.statProcessValues.error := FALSE;
   instCmCathodeAlignTableSuctionPlateVacuum.statProcessValues.interlockHomePos := TRUE;
   instCmCathodeAlignTableSuctionPlateVacuum.statProcessValues.interlockWorkPos := TRUE;
   instCmCathodeAlignTableSuctionPlateVacuum.statProcessValues.status := 16#7003;
   instCmCathodeAlignTableSuctionPlateVacuum.statProcessValues.interlockWarningWorkPos := FALSE;
   instCmCathodeAlignTableSuctionPlateVacuum.statProcessValues.interlockWarningHomePos := FALSE;
   instCmCathodeAlignTableSuctionPlateVacuum.statCurrentInputs.commandHomePos := FALSE;
   instCmCathodeAlignTableSuctionPlateVacuum.statCurrentInputs.commandWorkPos := FALSE;
   instCmCathodeAlignTableSuctionPlateVacuum.statCurrentInputs.reset := FALSE;
   instCmCathodeAlignTableSuctionPlateVacuum.statPreviousInputs.commandHomePos := FALSE;
   instCmCathodeAlignTableSuctionPlateVacuum.statPreviousInputs.commandWorkPos := FALSE;
   instCmCathodeAlignTableSuctionPlateVacuum.statPreviousInputs.reset := FALSE;
   instCmCathodeAlignTableSuctionPlateVacuum.statCurrentInterface.commandHomePos := FALSE;
   instCmCathodeAlignTableSuctionPlateVacuum.statCurrentInterface.commandWorkPos := FALSE;
   instCmCathodeAlignTableSuctionPlateVacuum.statCurrentInterface.reset := FALSE;
   instCmCathodeAlignTableSuctionPlateVacuum.statPreviousInterface.commandHomePos := FALSE;
   instCmCathodeAlignTableSuctionPlateVacuum.statPreviousInterface.commandWorkPos := FALSE;
   instCmCathodeAlignTableSuctionPlateVacuum.statPreviousInterface.reset := FALSE;
   instCmCathodeAlignTableSuctionPlateVacuum.statEmptyDiagnostics.status := 16#0000;
   instCmCathodeAlignTableSuctionPlateVacuum.statEmptyDiagnostics.subfunctionStatus := 16#0000;
   instCmCathodeAlignTableSuctionPlateVacuum.statEmptyDiagnostics.stateNumber := 0;
   instCmCathodeAlignTableSuctionPlateVacuum.instTimerReachPos.PT := T#0MS;
   instCmCathodeAlignTableSuctionPlateVacuum.instTimerReachPos.IN := FALSE;
   instCmCathodeAlignTableSuctionPlateVacuum.instTimerLeavePos.PT := T#0MS;
   instCmCathodeAlignTableSuctionPlateVacuum.instTimerLeavePos.IN := FALSE;
   instCmCathodeAlignTableSuctionPlateVacuum.instTimerDiscrepancyCheck.PT := T#0MS;
   instCmCathodeAlignTableSuctionPlateVacuum.instTimerDiscrepancyCheck.IN := FALSE;
   instCmCathodeAlignTableSuctionPlateVacuum.statDisableAlarms := FALSE;
   instCmCathodeAlignTableSuctionPlateVacuum.statDiagnostics.status := 16#7003;
   instCmCathodeAlignTableSuctionPlateVacuum.statDiagnostics.subfunctionStatus := 16#0000;
   instCmCathodeAlignTableSuctionPlateVacuum.statDiagnostics.stateNumber := 0;
   instCmCathodeAlignTableSuctionPlateVacuum.statEnablePrevious := TRUE;
   instCmCathodeAlignTableSuctionPlateVacuum.statFirstCall := FALSE;
   instCmCathodeAlignTableSuctionPlateVacuum.statResetPrevious := FALSE;
   instCmCathodeAlignTableSuctionPlateVacuum.statValid := TRUE;
   instCmCathodeAlignTableSuctionPlateVacuum.statBusy := TRUE;
   instCmCathodeAlignTableSuctionPlateVacuum.statError := FALSE;
   instCmCathodeAlignTableSuctionPlateVacuum.statInterlockWorkOff := FALSE;
   instCmCathodeAlignTableSuctionPlateVacuum.statInterlockHomeOff := FALSE;
   instCmCathodeAlignTableSuctionPlateVacuum.statFbState := 50;
   instCmCathodeAlignTableSuctionPlateVacuum.statFbStatePrevious := 50;
   instCmCathodeAlignTableSuctionPlateVacuum.statErrorUserCleared := FALSE;
   instCmCathodeAlignTableSuctionPlateVacuum.statErrorAutoCleared := FALSE;
   instCmCathodeAlignTableSuctionPlateVacuum.statErrorState := 16#0000;
   instCmCathodeAlignTableSuctionPlateVacuum.statDisablingCompleted := FALSE;
   instCmCathodeAlignTableSuctionPlateVacuum.statFeedbackHomePos := TRUE;
   instCmCathodeAlignTableSuctionPlateVacuum.statFeedbackWorkPos := FALSE;
   instCmCathodeGlassCleaning.enable := TRUE;
   instCmCathodeGlassCleaning.parentReferenceDesignator := WSTRING#'';
   instCmCathodeGlassCleaning.feedbackHomePos := FALSE;
   instCmCathodeGlassCleaning.feedbackWorkPos := FALSE;
   instCmCathodeGlassCleaning.enableManualCmds := TRUE;
   instCmCathodeGlassCleaning.interlockWorkPos := TRUE;
   instCmCathodeGlassCleaning.interlockHomePos := TRUE;
   instCmCathodeGlassCleaning.goToHomePos := FALSE;
   instCmCathodeGlassCleaning.goToWorkPos := FALSE;
   instCmCathodeGlassCleaning.statProcessValues.enable := TRUE;
   instCmCathodeGlassCleaning.statProcessValues.referenceDesignator := WSTRING#'GlassCleaning';
   instCmCathodeGlassCleaning.statProcessValues.commandHomePos := FALSE;
   instCmCathodeGlassCleaning.statProcessValues.commandWorkPos := FALSE;
   instCmCathodeGlassCleaning.statProcessValues.goToHomePos := FALSE;
   instCmCathodeGlassCleaning.statProcessValues.goToWorkPos := FALSE;
   instCmCathodeGlassCleaning.statProcessValues.inHomePos := FALSE;
   instCmCathodeGlassCleaning.statProcessValues.inWorkPos := FALSE;
   instCmCathodeGlassCleaning.statProcessValues.reset := FALSE;
   instCmCathodeGlassCleaning.statProcessValues.enableManualCmds := TRUE;
   instCmCathodeGlassCleaning.statProcessValues.error := FALSE;
   instCmCathodeGlassCleaning.statProcessValues.interlockHomePos := TRUE;
   instCmCathodeGlassCleaning.statProcessValues.interlockWorkPos := TRUE;
   instCmCathodeGlassCleaning.statProcessValues.status := 16#7003;
   instCmCathodeGlassCleaning.statProcessValues.interlockWarningWorkPos := FALSE;
   instCmCathodeGlassCleaning.statProcessValues.interlockWarningHomePos := FALSE;
   instCmCathodeGlassCleaning.statCurrentInputs.commandHomePos := FALSE;
   instCmCathodeGlassCleaning.statCurrentInputs.commandWorkPos := FALSE;
   instCmCathodeGlassCleaning.statCurrentInputs.reset := FALSE;
   instCmCathodeGlassCleaning.statPreviousInputs.commandHomePos := FALSE;
   instCmCathodeGlassCleaning.statPreviousInputs.commandWorkPos := FALSE;
   instCmCathodeGlassCleaning.statPreviousInputs.reset := FALSE;
   instCmCathodeGlassCleaning.statCurrentInterface.commandHomePos := FALSE;
   instCmCathodeGlassCleaning.statCurrentInterface.commandWorkPos := FALSE;
   instCmCathodeGlassCleaning.statCurrentInterface.reset := FALSE;
   instCmCathodeGlassCleaning.statPreviousInterface.commandHomePos := FALSE;
   instCmCathodeGlassCleaning.statPreviousInterface.commandWorkPos := FALSE;
   instCmCathodeGlassCleaning.statPreviousInterface.reset := FALSE;
   instCmCathodeGlassCleaning.statEmptyDiagnostics.status := 16#0000;
   instCmCathodeGlassCleaning.statEmptyDiagnostics.subfunctionStatus := 16#0000;
   instCmCathodeGlassCleaning.statEmptyDiagnostics.stateNumber := 0;
   instCmCathodeGlassCleaning.instTimerReachPos.PT := T#0MS;
   instCmCathodeGlassCleaning.instTimerReachPos.IN := FALSE;
   instCmCathodeGlassCleaning.instTimerLeavePos.PT := T#0MS;
   instCmCathodeGlassCleaning.instTimerLeavePos.IN := FALSE;
   instCmCathodeGlassCleaning.instTimerDiscrepancyCheck.PT := T#0MS;
   instCmCathodeGlassCleaning.instTimerDiscrepancyCheck.IN := FALSE;
   instCmCathodeGlassCleaning.statDisableAlarms := FALSE;
   instCmCathodeGlassCleaning.statDiagnostics.status := 16#7003;
   instCmCathodeGlassCleaning.statDiagnostics.subfunctionStatus := 16#0000;
   instCmCathodeGlassCleaning.statDiagnostics.stateNumber := 0;
   instCmCathodeGlassCleaning.statEnablePrevious := TRUE;
   instCmCathodeGlassCleaning.statFirstCall := FALSE;
   instCmCathodeGlassCleaning.statResetPrevious := FALSE;
   instCmCathodeGlassCleaning.statValid := TRUE;
   instCmCathodeGlassCleaning.statBusy := TRUE;
   instCmCathodeGlassCleaning.statError := FALSE;
   instCmCathodeGlassCleaning.statInterlockWorkOff := FALSE;
   instCmCathodeGlassCleaning.statInterlockHomeOff := FALSE;
   instCmCathodeGlassCleaning.statFbState := 50;
   instCmCathodeGlassCleaning.statFbStatePrevious := 50;
   instCmCathodeGlassCleaning.statErrorUserCleared := FALSE;
   instCmCathodeGlassCleaning.statErrorAutoCleared := FALSE;
   instCmCathodeGlassCleaning.statErrorState := 16#0000;
   instCmCathodeGlassCleaning.statDisablingCompleted := FALSE;
   instCmCathodeGlassCleaning.statFeedbackHomePos := FALSE;
   instCmCathodeGlassCleaning.statFeedbackWorkPos := FALSE;
   instCmCathodeNgPnpUpDown.enable := TRUE;
   instCmCathodeNgPnpUpDown.parentReferenceDesignator := WSTRING#'';
   instCmCathodeNgPnpUpDown.feedbackHomePos := FALSE;
   instCmCathodeNgPnpUpDown.feedbackWorkPos := TRUE;
   instCmCathodeNgPnpUpDown.enableManualCmds := TRUE;
   instCmCathodeNgPnpUpDown.interlockWorkPos := FALSE;
   instCmCathodeNgPnpUpDown.interlockHomePos := TRUE;
   instCmCathodeNgPnpUpDown.goToHomePos := FALSE;
   instCmCathodeNgPnpUpDown.goToWorkPos := FALSE;
   instCmCathodeNgPnpUpDown.statProcessValues.enable := TRUE;
   instCmCathodeNgPnpUpDown.statProcessValues.referenceDesignator := WSTRING#'NgPnpUpDown';
   instCmCathodeNgPnpUpDown.statProcessValues.commandHomePos := FALSE;
   instCmCathodeNgPnpUpDown.statProcessValues.commandWorkPos := FALSE;
   instCmCathodeNgPnpUpDown.statProcessValues.goToHomePos := FALSE;
   instCmCathodeNgPnpUpDown.statProcessValues.goToWorkPos := FALSE;
   instCmCathodeNgPnpUpDown.statProcessValues.inHomePos := FALSE;
   instCmCathodeNgPnpUpDown.statProcessValues.inWorkPos := FALSE;
   instCmCathodeNgPnpUpDown.statProcessValues.reset := FALSE;
   instCmCathodeNgPnpUpDown.statProcessValues.enableManualCmds := TRUE;
   instCmCathodeNgPnpUpDown.statProcessValues.error := FALSE;
   instCmCathodeNgPnpUpDown.statProcessValues.interlockHomePos := TRUE;
   instCmCathodeNgPnpUpDown.statProcessValues.interlockWorkPos := FALSE;
   instCmCathodeNgPnpUpDown.statProcessValues.status := 16#7101;
   instCmCathodeNgPnpUpDown.statProcessValues.interlockWarningWorkPos := FALSE;
   instCmCathodeNgPnpUpDown.statProcessValues.interlockWarningHomePos := FALSE;
   instCmCathodeNgPnpUpDown.statCurrentInputs.commandHomePos := FALSE;
   instCmCathodeNgPnpUpDown.statCurrentInputs.commandWorkPos := FALSE;
   instCmCathodeNgPnpUpDown.statCurrentInputs.reset := FALSE;
   instCmCathodeNgPnpUpDown.statPreviousInputs.commandHomePos := FALSE;
   instCmCathodeNgPnpUpDown.statPreviousInputs.commandWorkPos := FALSE;
   instCmCathodeNgPnpUpDown.statPreviousInputs.reset := FALSE;
   instCmCathodeNgPnpUpDown.statCurrentInterface.commandHomePos := FALSE;
   instCmCathodeNgPnpUpDown.statCurrentInterface.commandWorkPos := FALSE;
   instCmCathodeNgPnpUpDown.statCurrentInterface.reset := FALSE;
   instCmCathodeNgPnpUpDown.statPreviousInterface.commandHomePos := FALSE;
   instCmCathodeNgPnpUpDown.statPreviousInterface.commandWorkPos := FALSE;
   instCmCathodeNgPnpUpDown.statPreviousInterface.reset := FALSE;
   instCmCathodeNgPnpUpDown.statEmptyDiagnostics.status := 16#0000;
   instCmCathodeNgPnpUpDown.statEmptyDiagnostics.subfunctionStatus := 16#0000;
   instCmCathodeNgPnpUpDown.statEmptyDiagnostics.stateNumber := 0;
   instCmCathodeNgPnpUpDown.instTimerReachPos.PT := T#0MS;
   instCmCathodeNgPnpUpDown.instTimerReachPos.IN := FALSE;
   instCmCathodeNgPnpUpDown.instTimerLeavePos.PT := T#0MS;
   instCmCathodeNgPnpUpDown.instTimerLeavePos.IN := FALSE;
   instCmCathodeNgPnpUpDown.instTimerDiscrepancyCheck.PT := T#0MS;
   instCmCathodeNgPnpUpDown.instTimerDiscrepancyCheck.IN := FALSE;
   instCmCathodeNgPnpUpDown.statDisableAlarms := FALSE;
   instCmCathodeNgPnpUpDown.statDiagnostics.status := 16#7003;
   instCmCathodeNgPnpUpDown.statDiagnostics.subfunctionStatus := 16#0000;
   instCmCathodeNgPnpUpDown.statDiagnostics.stateNumber := 0;
   instCmCathodeNgPnpUpDown.statEnablePrevious := TRUE;
   instCmCathodeNgPnpUpDown.statFirstCall := FALSE;
   instCmCathodeNgPnpUpDown.statResetPrevious := FALSE;
   instCmCathodeNgPnpUpDown.statValid := TRUE;
   instCmCathodeNgPnpUpDown.statBusy := TRUE;
   instCmCathodeNgPnpUpDown.statError := FALSE;
   instCmCathodeNgPnpUpDown.statInterlockWorkOff := FALSE;
   instCmCathodeNgPnpUpDown.statInterlockHomeOff := FALSE;
   instCmCathodeNgPnpUpDown.statFbState := 50;
   instCmCathodeNgPnpUpDown.statFbStatePrevious := 50;
   instCmCathodeNgPnpUpDown.statErrorUserCleared := FALSE;
   instCmCathodeNgPnpUpDown.statErrorAutoCleared := FALSE;
   instCmCathodeNgPnpUpDown.statErrorState := 16#0000;
   instCmCathodeNgPnpUpDown.statDisablingCompleted := FALSE;
   instCmCathodeNgPnpUpDown.statFeedbackHomePos := FALSE;
   instCmCathodeNgPnpUpDown.statFeedbackWorkPos := TRUE;
   instCmCathodeNgPnp1stFwdBwd.enable := TRUE;
   instCmCathodeNgPnp1stFwdBwd.parentReferenceDesignator := WSTRING#'';
   instCmCathodeNgPnp1stFwdBwd.feedbackHomePos := TRUE;
   instCmCathodeNgPnp1stFwdBwd.feedbackWorkPos := FALSE;
   instCmCathodeNgPnp1stFwdBwd.enableManualCmds := TRUE;
   instCmCathodeNgPnp1stFwdBwd.interlockWorkPos := FALSE;
   instCmCathodeNgPnp1stFwdBwd.interlockHomePos := TRUE;
   instCmCathodeNgPnp1stFwdBwd.goToHomePos := FALSE;
   instCmCathodeNgPnp1stFwdBwd.goToWorkPos := FALSE;
   instCmCathodeNgPnp1stFwdBwd.statProcessValues.enable := TRUE;
   instCmCathodeNgPnp1stFwdBwd.statProcessValues.referenceDesignator := WSTRING#'NgPnp1stFwdBwd';
   instCmCathodeNgPnp1stFwdBwd.statProcessValues.commandHomePos := FALSE;
   instCmCathodeNgPnp1stFwdBwd.statProcessValues.commandWorkPos := FALSE;
   instCmCathodeNgPnp1stFwdBwd.statProcessValues.goToHomePos := FALSE;
   instCmCathodeNgPnp1stFwdBwd.statProcessValues.goToWorkPos := FALSE;
   instCmCathodeNgPnp1stFwdBwd.statProcessValues.inHomePos := TRUE;
   instCmCathodeNgPnp1stFwdBwd.statProcessValues.inWorkPos := FALSE;
   instCmCathodeNgPnp1stFwdBwd.statProcessValues.reset := FALSE;
   instCmCathodeNgPnp1stFwdBwd.statProcessValues.enableManualCmds := TRUE;
   instCmCathodeNgPnp1stFwdBwd.statProcessValues.error := FALSE;
   instCmCathodeNgPnp1stFwdBwd.statProcessValues.interlockHomePos := TRUE;
   instCmCathodeNgPnp1stFwdBwd.statProcessValues.interlockWorkPos := FALSE;
   instCmCathodeNgPnp1stFwdBwd.statProcessValues.status := 16#7101;
   instCmCathodeNgPnp1stFwdBwd.statProcessValues.interlockWarningWorkPos := FALSE;
   instCmCathodeNgPnp1stFwdBwd.statProcessValues.interlockWarningHomePos := FALSE;
   instCmCathodeNgPnp1stFwdBwd.statCurrentInputs.commandHomePos := FALSE;
   instCmCathodeNgPnp1stFwdBwd.statCurrentInputs.commandWorkPos := FALSE;
   instCmCathodeNgPnp1stFwdBwd.statCurrentInputs.reset := FALSE;
   instCmCathodeNgPnp1stFwdBwd.statPreviousInputs.commandHomePos := FALSE;
   instCmCathodeNgPnp1stFwdBwd.statPreviousInputs.commandWorkPos := FALSE;
   instCmCathodeNgPnp1stFwdBwd.statPreviousInputs.reset := FALSE;
   instCmCathodeNgPnp1stFwdBwd.statCurrentInterface.commandHomePos := FALSE;
   instCmCathodeNgPnp1stFwdBwd.statCurrentInterface.commandWorkPos := FALSE;
   instCmCathodeNgPnp1stFwdBwd.statCurrentInterface.reset := FALSE;
   instCmCathodeNgPnp1stFwdBwd.statPreviousInterface.commandHomePos := FALSE;
   instCmCathodeNgPnp1stFwdBwd.statPreviousInterface.commandWorkPos := FALSE;
   instCmCathodeNgPnp1stFwdBwd.statPreviousInterface.reset := FALSE;
   instCmCathodeNgPnp1stFwdBwd.statEmptyDiagnostics.status := 16#0000;
   instCmCathodeNgPnp1stFwdBwd.statEmptyDiagnostics.subfunctionStatus := 16#0000;
   instCmCathodeNgPnp1stFwdBwd.statEmptyDiagnostics.stateNumber := 0;
   instCmCathodeNgPnp1stFwdBwd.instTimerReachPos.PT := T#0MS;
   instCmCathodeNgPnp1stFwdBwd.instTimerReachPos.IN := FALSE;
   instCmCathodeNgPnp1stFwdBwd.instTimerLeavePos.PT := T#0MS;
   instCmCathodeNgPnp1stFwdBwd.instTimerLeavePos.IN := FALSE;
   instCmCathodeNgPnp1stFwdBwd.instTimerDiscrepancyCheck.PT := T#0MS;
   instCmCathodeNgPnp1stFwdBwd.instTimerDiscrepancyCheck.IN := FALSE;
   instCmCathodeNgPnp1stFwdBwd.statDisableAlarms := FALSE;
   instCmCathodeNgPnp1stFwdBwd.statDiagnostics.status := 16#7003;
   instCmCathodeNgPnp1stFwdBwd.statDiagnostics.subfunctionStatus := 16#0000;
   instCmCathodeNgPnp1stFwdBwd.statDiagnostics.stateNumber := 0;
   instCmCathodeNgPnp1stFwdBwd.statEnablePrevious := TRUE;
   instCmCathodeNgPnp1stFwdBwd.statFirstCall := FALSE;
   instCmCathodeNgPnp1stFwdBwd.statResetPrevious := FALSE;
   instCmCathodeNgPnp1stFwdBwd.statValid := TRUE;
   instCmCathodeNgPnp1stFwdBwd.statBusy := TRUE;
   instCmCathodeNgPnp1stFwdBwd.statError := FALSE;
   instCmCathodeNgPnp1stFwdBwd.statInterlockWorkOff := FALSE;
   instCmCathodeNgPnp1stFwdBwd.statInterlockHomeOff := FALSE;
   instCmCathodeNgPnp1stFwdBwd.statFbState := 50;
   instCmCathodeNgPnp1stFwdBwd.statFbStatePrevious := 50;
   instCmCathodeNgPnp1stFwdBwd.statErrorUserCleared := FALSE;
   instCmCathodeNgPnp1stFwdBwd.statErrorAutoCleared := FALSE;
   instCmCathodeNgPnp1stFwdBwd.statErrorState := 16#0000;
   instCmCathodeNgPnp1stFwdBwd.statDisablingCompleted := FALSE;
   instCmCathodeNgPnp1stFwdBwd.statFeedbackHomePos := TRUE;
   instCmCathodeNgPnp1stFwdBwd.statFeedbackWorkPos := FALSE;
   instCmCathodeNgPnp2ndFwdBwd.enable := TRUE;
   instCmCathodeNgPnp2ndFwdBwd.parentReferenceDesignator := WSTRING#'';
   instCmCathodeNgPnp2ndFwdBwd.feedbackHomePos := TRUE;
   instCmCathodeNgPnp2ndFwdBwd.feedbackWorkPos := FALSE;
   instCmCathodeNgPnp2ndFwdBwd.enableManualCmds := TRUE;
   instCmCathodeNgPnp2ndFwdBwd.interlockWorkPos := FALSE;
   instCmCathodeNgPnp2ndFwdBwd.interlockHomePos := FALSE;
   instCmCathodeNgPnp2ndFwdBwd.goToHomePos := FALSE;
   instCmCathodeNgPnp2ndFwdBwd.goToWorkPos := FALSE;
   instCmCathodeNgPnp2ndFwdBwd.statProcessValues.enable := TRUE;
   instCmCathodeNgPnp2ndFwdBwd.statProcessValues.referenceDesignator := WSTRING#'NgPnp2ndFwdBwd';
   instCmCathodeNgPnp2ndFwdBwd.statProcessValues.commandHomePos := FALSE;
   instCmCathodeNgPnp2ndFwdBwd.statProcessValues.commandWorkPos := FALSE;
   instCmCathodeNgPnp2ndFwdBwd.statProcessValues.goToHomePos := FALSE;
   instCmCathodeNgPnp2ndFwdBwd.statProcessValues.goToWorkPos := FALSE;
   instCmCathodeNgPnp2ndFwdBwd.statProcessValues.inHomePos := FALSE;
   instCmCathodeNgPnp2ndFwdBwd.statProcessValues.inWorkPos := FALSE;
   instCmCathodeNgPnp2ndFwdBwd.statProcessValues.reset := FALSE;
   instCmCathodeNgPnp2ndFwdBwd.statProcessValues.enableManualCmds := TRUE;
   instCmCathodeNgPnp2ndFwdBwd.statProcessValues.error := FALSE;
   instCmCathodeNgPnp2ndFwdBwd.statProcessValues.interlockHomePos := FALSE;
   instCmCathodeNgPnp2ndFwdBwd.statProcessValues.interlockWorkPos := FALSE;
   instCmCathodeNgPnp2ndFwdBwd.statProcessValues.status := 16#7100;
   instCmCathodeNgPnp2ndFwdBwd.statProcessValues.interlockWarningWorkPos := FALSE;
   instCmCathodeNgPnp2ndFwdBwd.statProcessValues.interlockWarningHomePos := FALSE;
   instCmCathodeNgPnp2ndFwdBwd.statCurrentInputs.commandHomePos := FALSE;
   instCmCathodeNgPnp2ndFwdBwd.statCurrentInputs.commandWorkPos := FALSE;
   instCmCathodeNgPnp2ndFwdBwd.statCurrentInputs.reset := FALSE;
   instCmCathodeNgPnp2ndFwdBwd.statPreviousInputs.commandHomePos := FALSE;
   instCmCathodeNgPnp2ndFwdBwd.statPreviousInputs.commandWorkPos := FALSE;
   instCmCathodeNgPnp2ndFwdBwd.statPreviousInputs.reset := FALSE;
   instCmCathodeNgPnp2ndFwdBwd.statCurrentInterface.commandHomePos := FALSE;
   instCmCathodeNgPnp2ndFwdBwd.statCurrentInterface.commandWorkPos := FALSE;
   instCmCathodeNgPnp2ndFwdBwd.statCurrentInterface.reset := FALSE;
   instCmCathodeNgPnp2ndFwdBwd.statPreviousInterface.commandHomePos := FALSE;
   instCmCathodeNgPnp2ndFwdBwd.statPreviousInterface.commandWorkPos := FALSE;
   instCmCathodeNgPnp2ndFwdBwd.statPreviousInterface.reset := FALSE;
   instCmCathodeNgPnp2ndFwdBwd.statEmptyDiagnostics.status := 16#0000;
   instCmCathodeNgPnp2ndFwdBwd.statEmptyDiagnostics.subfunctionStatus := 16#0000;
   instCmCathodeNgPnp2ndFwdBwd.statEmptyDiagnostics.stateNumber := 0;
   instCmCathodeNgPnp2ndFwdBwd.instTimerReachPos.PT := T#0MS;
   instCmCathodeNgPnp2ndFwdBwd.instTimerReachPos.IN := FALSE;
   instCmCathodeNgPnp2ndFwdBwd.instTimerLeavePos.PT := T#0MS;
   instCmCathodeNgPnp2ndFwdBwd.instTimerLeavePos.IN := FALSE;
   instCmCathodeNgPnp2ndFwdBwd.instTimerDiscrepancyCheck.PT := T#0MS;
   instCmCathodeNgPnp2ndFwdBwd.instTimerDiscrepancyCheck.IN := FALSE;
   instCmCathodeNgPnp2ndFwdBwd.statDisableAlarms := FALSE;
   instCmCathodeNgPnp2ndFwdBwd.statDiagnostics.status := 16#7003;
   instCmCathodeNgPnp2ndFwdBwd.statDiagnostics.subfunctionStatus := 16#0000;
   instCmCathodeNgPnp2ndFwdBwd.statDiagnostics.stateNumber := 0;
   instCmCathodeNgPnp2ndFwdBwd.statEnablePrevious := TRUE;
   instCmCathodeNgPnp2ndFwdBwd.statFirstCall := FALSE;
   instCmCathodeNgPnp2ndFwdBwd.statResetPrevious := FALSE;
   instCmCathodeNgPnp2ndFwdBwd.statValid := TRUE;
   instCmCathodeNgPnp2ndFwdBwd.statBusy := TRUE;
   instCmCathodeNgPnp2ndFwdBwd.statError := FALSE;
   instCmCathodeNgPnp2ndFwdBwd.statInterlockWorkOff := FALSE;
   instCmCathodeNgPnp2ndFwdBwd.statInterlockHomeOff := FALSE;
   instCmCathodeNgPnp2ndFwdBwd.statFbState := 50;
   instCmCathodeNgPnp2ndFwdBwd.statFbStatePrevious := 50;
   instCmCathodeNgPnp2ndFwdBwd.statErrorUserCleared := FALSE;
   instCmCathodeNgPnp2ndFwdBwd.statErrorAutoCleared := FALSE;
   instCmCathodeNgPnp2ndFwdBwd.statErrorState := 16#0000;
   instCmCathodeNgPnp2ndFwdBwd.statDisablingCompleted := FALSE;
   instCmCathodeNgPnp2ndFwdBwd.statFeedbackHomePos := TRUE;
   instCmCathodeNgPnp2ndFwdBwd.statFeedbackWorkPos := FALSE;
   instCmCathodeMaintenanceMovingFixFwdBwd.enable := TRUE;
   instCmCathodeMaintenanceMovingFixFwdBwd.parentReferenceDesignator := WSTRING#'';
   instCmCathodeMaintenanceMovingFixFwdBwd.feedbackHomePos := FALSE;
   instCmCathodeMaintenanceMovingFixFwdBwd.feedbackWorkPos := TRUE;
   instCmCathodeMaintenanceMovingFixFwdBwd.enableManualCmds := TRUE;
   instCmCathodeMaintenanceMovingFixFwdBwd.interlockWorkPos := TRUE;
   instCmCathodeMaintenanceMovingFixFwdBwd.interlockHomePos := TRUE;
   instCmCathodeMaintenanceMovingFixFwdBwd.goToHomePos := FALSE;
   instCmCathodeMaintenanceMovingFixFwdBwd.goToWorkPos := FALSE;
   instCmCathodeMaintenanceMovingFixFwdBwd.statProcessValues.enable := TRUE;
   instCmCathodeMaintenanceMovingFixFwdBwd.statProcessValues.referenceDesignator := WSTRING#'MaintenanceFix';
   instCmCathodeMaintenanceMovingFixFwdBwd.statProcessValues.commandHomePos := FALSE;
   instCmCathodeMaintenanceMovingFixFwdBwd.statProcessValues.commandWorkPos := FALSE;
   instCmCathodeMaintenanceMovingFixFwdBwd.statProcessValues.goToHomePos := FALSE;
   instCmCathodeMaintenanceMovingFixFwdBwd.statProcessValues.goToWorkPos := FALSE;
   instCmCathodeMaintenanceMovingFixFwdBwd.statProcessValues.inHomePos := FALSE;
   instCmCathodeMaintenanceMovingFixFwdBwd.statProcessValues.inWorkPos := TRUE;
   instCmCathodeMaintenanceMovingFixFwdBwd.statProcessValues.reset := FALSE;
   instCmCathodeMaintenanceMovingFixFwdBwd.statProcessValues.enableManualCmds := TRUE;
   instCmCathodeMaintenanceMovingFixFwdBwd.statProcessValues.error := FALSE;
   instCmCathodeMaintenanceMovingFixFwdBwd.statProcessValues.interlockHomePos := TRUE;
   instCmCathodeMaintenanceMovingFixFwdBwd.statProcessValues.interlockWorkPos := TRUE;
   instCmCathodeMaintenanceMovingFixFwdBwd.statProcessValues.status := 16#7003;
   instCmCathodeMaintenanceMovingFixFwdBwd.statProcessValues.interlockWarningWorkPos := FALSE;
   instCmCathodeMaintenanceMovingFixFwdBwd.statProcessValues.interlockWarningHomePos := FALSE;
   instCmCathodeMaintenanceMovingFixFwdBwd.statCurrentInputs.commandHomePos := FALSE;
   instCmCathodeMaintenanceMovingFixFwdBwd.statCurrentInputs.commandWorkPos := FALSE;
   instCmCathodeMaintenanceMovingFixFwdBwd.statCurrentInputs.reset := FALSE;
   instCmCathodeMaintenanceMovingFixFwdBwd.statPreviousInputs.commandHomePos := FALSE;
   instCmCathodeMaintenanceMovingFixFwdBwd.statPreviousInputs.commandWorkPos := FALSE;
   instCmCathodeMaintenanceMovingFixFwdBwd.statPreviousInputs.reset := FALSE;
   instCmCathodeMaintenanceMovingFixFwdBwd.statCurrentInterface.commandHomePos := FALSE;
   instCmCathodeMaintenanceMovingFixFwdBwd.statCurrentInterface.commandWorkPos := FALSE;
   instCmCathodeMaintenanceMovingFixFwdBwd.statCurrentInterface.reset := FALSE;
   instCmCathodeMaintenanceMovingFixFwdBwd.statPreviousInterface.commandHomePos := FALSE;
   instCmCathodeMaintenanceMovingFixFwdBwd.statPreviousInterface.commandWorkPos := FALSE;
   instCmCathodeMaintenanceMovingFixFwdBwd.statPreviousInterface.reset := FALSE;
   instCmCathodeMaintenanceMovingFixFwdBwd.statEmptyDiagnostics.status := 16#0000;
   instCmCathodeMaintenanceMovingFixFwdBwd.statEmptyDiagnostics.subfunctionStatus := 16#0000;
   instCmCathodeMaintenanceMovingFixFwdBwd.statEmptyDiagnostics.stateNumber := 0;
   instCmCathodeMaintenanceMovingFixFwdBwd.instTimerReachPos.PT := T#0MS;
   instCmCathodeMaintenanceMovingFixFwdBwd.instTimerReachPos.IN := FALSE;
   instCmCathodeMaintenanceMovingFixFwdBwd.instTimerLeavePos.PT := T#0MS;
   instCmCathodeMaintenanceMovingFixFwdBwd.instTimerLeavePos.IN := FALSE;
   instCmCathodeMaintenanceMovingFixFwdBwd.instTimerDiscrepancyCheck.PT := T#0MS;
   instCmCathodeMaintenanceMovingFixFwdBwd.instTimerDiscrepancyCheck.IN := FALSE;
   instCmCathodeMaintenanceMovingFixFwdBwd.statDisableAlarms := FALSE;
   instCmCathodeMaintenanceMovingFixFwdBwd.statDiagnostics.status := 16#7003;
   instCmCathodeMaintenanceMovingFixFwdBwd.statDiagnostics.subfunctionStatus := 16#0000;
   instCmCathodeMaintenanceMovingFixFwdBwd.statDiagnostics.stateNumber := 0;
   instCmCathodeMaintenanceMovingFixFwdBwd.statEnablePrevious := TRUE;
   instCmCathodeMaintenanceMovingFixFwdBwd.statFirstCall := FALSE;
   instCmCathodeMaintenanceMovingFixFwdBwd.statResetPrevious := FALSE;
   instCmCathodeMaintenanceMovingFixFwdBwd.statValid := TRUE;
   instCmCathodeMaintenanceMovingFixFwdBwd.statBusy := TRUE;
   instCmCathodeMaintenanceMovingFixFwdBwd.statError := FALSE;
   instCmCathodeMaintenanceMovingFixFwdBwd.statInterlockWorkOff := FALSE;
   instCmCathodeMaintenanceMovingFixFwdBwd.statInterlockHomeOff := FALSE;
   instCmCathodeMaintenanceMovingFixFwdBwd.statFbState := 50;
   instCmCathodeMaintenanceMovingFixFwdBwd.statFbStatePrevious := 50;
   instCmCathodeMaintenanceMovingFixFwdBwd.statErrorUserCleared := FALSE;
   instCmCathodeMaintenanceMovingFixFwdBwd.statErrorAutoCleared := FALSE;
   instCmCathodeMaintenanceMovingFixFwdBwd.statErrorState := 16#0000;
   instCmCathodeMaintenanceMovingFixFwdBwd.statDisablingCompleted := FALSE;
   instCmCathodeMaintenanceMovingFixFwdBwd.statFeedbackHomePos := FALSE;
   instCmCathodeMaintenanceMovingFixFwdBwd.statFeedbackWorkPos := TRUE;
   instCmCathodeNgBoxLiftUpDown.enable := TRUE;
   instCmCathodeNgBoxLiftUpDown.parentReferenceDesignator := WSTRING#'';
   instCmCathodeNgBoxLiftUpDown.feedbackHomePos := TRUE;
   instCmCathodeNgBoxLiftUpDown.feedbackWorkPos := FALSE;
   instCmCathodeNgBoxLiftUpDown.enableManualCmds := TRUE;
   instCmCathodeNgBoxLiftUpDown.interlockWorkPos := FALSE;
   instCmCathodeNgBoxLiftUpDown.interlockHomePos := TRUE;
   instCmCathodeNgBoxLiftUpDown.goToHomePos := FALSE;
   instCmCathodeNgBoxLiftUpDown.goToWorkPos := FALSE;
   instCmCathodeNgBoxLiftUpDown.statProcessValues.enable := TRUE;
   instCmCathodeNgBoxLiftUpDown.statProcessValues.referenceDesignator := WSTRING#'NgBoxLiftUpDown';
   instCmCathodeNgBoxLiftUpDown.statProcessValues.commandHomePos := FALSE;
   instCmCathodeNgBoxLiftUpDown.statProcessValues.commandWorkPos := FALSE;
   instCmCathodeNgBoxLiftUpDown.statProcessValues.goToHomePos := FALSE;
   instCmCathodeNgBoxLiftUpDown.statProcessValues.goToWorkPos := FALSE;
   instCmCathodeNgBoxLiftUpDown.statProcessValues.inHomePos := TRUE;
   instCmCathodeNgBoxLiftUpDown.statProcessValues.inWorkPos := FALSE;
   instCmCathodeNgBoxLiftUpDown.statProcessValues.reset := FALSE;
   instCmCathodeNgBoxLiftUpDown.statProcessValues.enableManualCmds := TRUE;
   instCmCathodeNgBoxLiftUpDown.statProcessValues.error := FALSE;
   instCmCathodeNgBoxLiftUpDown.statProcessValues.interlockHomePos := TRUE;
   instCmCathodeNgBoxLiftUpDown.statProcessValues.interlockWorkPos := FALSE;
   instCmCathodeNgBoxLiftUpDown.statProcessValues.status := 16#7101;
   instCmCathodeNgBoxLiftUpDown.statProcessValues.interlockWarningWorkPos := FALSE;
   instCmCathodeNgBoxLiftUpDown.statProcessValues.interlockWarningHomePos := FALSE;
   instCmCathodeNgBoxLiftUpDown.statCurrentInputs.commandHomePos := FALSE;
   instCmCathodeNgBoxLiftUpDown.statCurrentInputs.commandWorkPos := FALSE;
   instCmCathodeNgBoxLiftUpDown.statCurrentInputs.reset := FALSE;
   instCmCathodeNgBoxLiftUpDown.statPreviousInputs.commandHomePos := FALSE;
   instCmCathodeNgBoxLiftUpDown.statPreviousInputs.commandWorkPos := FALSE;
   instCmCathodeNgBoxLiftUpDown.statPreviousInputs.reset := FALSE;
   instCmCathodeNgBoxLiftUpDown.statCurrentInterface.commandHomePos := FALSE;
   instCmCathodeNgBoxLiftUpDown.statCurrentInterface.commandWorkPos := FALSE;
   instCmCathodeNgBoxLiftUpDown.statCurrentInterface.reset := FALSE;
   instCmCathodeNgBoxLiftUpDown.statPreviousInterface.commandHomePos := FALSE;
   instCmCathodeNgBoxLiftUpDown.statPreviousInterface.commandWorkPos := FALSE;
   instCmCathodeNgBoxLiftUpDown.statPreviousInterface.reset := FALSE;
   instCmCathodeNgBoxLiftUpDown.statEmptyDiagnostics.status := 16#0000;
   instCmCathodeNgBoxLiftUpDown.statEmptyDiagnostics.subfunctionStatus := 16#0000;
   instCmCathodeNgBoxLiftUpDown.statEmptyDiagnostics.stateNumber := 0;
   instCmCathodeNgBoxLiftUpDown.instTimerReachPos.PT := T#0MS;
   instCmCathodeNgBoxLiftUpDown.instTimerReachPos.IN := FALSE;
   instCmCathodeNgBoxLiftUpDown.instTimerLeavePos.PT := T#0MS;
   instCmCathodeNgBoxLiftUpDown.instTimerLeavePos.IN := FALSE;
   instCmCathodeNgBoxLiftUpDown.instTimerDiscrepancyCheck.PT := T#0MS;
   instCmCathodeNgBoxLiftUpDown.instTimerDiscrepancyCheck.IN := FALSE;
   instCmCathodeNgBoxLiftUpDown.statDisableAlarms := FALSE;
   instCmCathodeNgBoxLiftUpDown.statDiagnostics.status := 16#7003;
   instCmCathodeNgBoxLiftUpDown.statDiagnostics.subfunctionStatus := 16#0000;
   instCmCathodeNgBoxLiftUpDown.statDiagnostics.stateNumber := 0;
   instCmCathodeNgBoxLiftUpDown.statEnablePrevious := TRUE;
   instCmCathodeNgBoxLiftUpDown.statFirstCall := FALSE;
   instCmCathodeNgBoxLiftUpDown.statResetPrevious := FALSE;
   instCmCathodeNgBoxLiftUpDown.statValid := TRUE;
   instCmCathodeNgBoxLiftUpDown.statBusy := TRUE;
   instCmCathodeNgBoxLiftUpDown.statError := FALSE;
   instCmCathodeNgBoxLiftUpDown.statInterlockWorkOff := FALSE;
   instCmCathodeNgBoxLiftUpDown.statInterlockHomeOff := FALSE;
   instCmCathodeNgBoxLiftUpDown.statFbState := 50;
   instCmCathodeNgBoxLiftUpDown.statFbStatePrevious := 50;
   instCmCathodeNgBoxLiftUpDown.statErrorUserCleared := FALSE;
   instCmCathodeNgBoxLiftUpDown.statErrorAutoCleared := FALSE;
   instCmCathodeNgBoxLiftUpDown.statErrorState := 16#0000;
   instCmCathodeNgBoxLiftUpDown.statDisablingCompleted := FALSE;
   instCmCathodeNgBoxLiftUpDown.statFeedbackHomePos := TRUE;
   instCmCathodeNgBoxLiftUpDown.statFeedbackWorkPos := FALSE;
   instCmCathodeNgBoxLockUpDown.enable := TRUE;
   instCmCathodeNgBoxLockUpDown.parentReferenceDesignator := WSTRING#'';
   instCmCathodeNgBoxLockUpDown.feedbackHomePos := TRUE;
   instCmCathodeNgBoxLockUpDown.feedbackWorkPos := FALSE;
   instCmCathodeNgBoxLockUpDown.enableManualCmds := TRUE;
   instCmCathodeNgBoxLockUpDown.interlockWorkPos := TRUE;
   instCmCathodeNgBoxLockUpDown.interlockHomePos := TRUE;
   instCmCathodeNgBoxLockUpDown.goToHomePos := FALSE;
   instCmCathodeNgBoxLockUpDown.goToWorkPos := FALSE;
   instCmCathodeNgBoxLockUpDown.statProcessValues.enable := TRUE;
   instCmCathodeNgBoxLockUpDown.statProcessValues.referenceDesignator := WSTRING#'NgBoxLockUpDown';
   instCmCathodeNgBoxLockUpDown.statProcessValues.commandHomePos := FALSE;
   instCmCathodeNgBoxLockUpDown.statProcessValues.commandWorkPos := FALSE;
   instCmCathodeNgBoxLockUpDown.statProcessValues.goToHomePos := FALSE;
   instCmCathodeNgBoxLockUpDown.statProcessValues.goToWorkPos := FALSE;
   instCmCathodeNgBoxLockUpDown.statProcessValues.inHomePos := TRUE;
   instCmCathodeNgBoxLockUpDown.statProcessValues.inWorkPos := FALSE;
   instCmCathodeNgBoxLockUpDown.statProcessValues.reset := FALSE;
   instCmCathodeNgBoxLockUpDown.statProcessValues.enableManualCmds := TRUE;
   instCmCathodeNgBoxLockUpDown.statProcessValues.error := FALSE;
   instCmCathodeNgBoxLockUpDown.statProcessValues.interlockHomePos := TRUE;
   instCmCathodeNgBoxLockUpDown.statProcessValues.interlockWorkPos := TRUE;
   instCmCathodeNgBoxLockUpDown.statProcessValues.status := 16#7003;
   instCmCathodeNgBoxLockUpDown.statProcessValues.interlockWarningWorkPos := FALSE;
   instCmCathodeNgBoxLockUpDown.statProcessValues.interlockWarningHomePos := FALSE;
   instCmCathodeNgBoxLockUpDown.statCurrentInputs.commandHomePos := FALSE;
   instCmCathodeNgBoxLockUpDown.statCurrentInputs.commandWorkPos := FALSE;
   instCmCathodeNgBoxLockUpDown.statCurrentInputs.reset := FALSE;
   instCmCathodeNgBoxLockUpDown.statPreviousInputs.commandHomePos := FALSE;
   instCmCathodeNgBoxLockUpDown.statPreviousInputs.commandWorkPos := FALSE;
   instCmCathodeNgBoxLockUpDown.statPreviousInputs.reset := FALSE;
   instCmCathodeNgBoxLockUpDown.statCurrentInterface.commandHomePos := FALSE;
   instCmCathodeNgBoxLockUpDown.statCurrentInterface.commandWorkPos := FALSE;
   instCmCathodeNgBoxLockUpDown.statCurrentInterface.reset := FALSE;
   instCmCathodeNgBoxLockUpDown.statPreviousInterface.commandHomePos := FALSE;
   instCmCathodeNgBoxLockUpDown.statPreviousInterface.commandWorkPos := FALSE;
   instCmCathodeNgBoxLockUpDown.statPreviousInterface.reset := FALSE;
   instCmCathodeNgBoxLockUpDown.statEmptyDiagnostics.status := 16#0000;
   instCmCathodeNgBoxLockUpDown.statEmptyDiagnostics.subfunctionStatus := 16#0000;
   instCmCathodeNgBoxLockUpDown.statEmptyDiagnostics.stateNumber := 0;
   instCmCathodeNgBoxLockUpDown.instTimerReachPos.PT := T#0MS;
   instCmCathodeNgBoxLockUpDown.instTimerReachPos.IN := FALSE;
   instCmCathodeNgBoxLockUpDown.instTimerLeavePos.PT := T#0MS;
   instCmCathodeNgBoxLockUpDown.instTimerLeavePos.IN := FALSE;
   instCmCathodeNgBoxLockUpDown.instTimerDiscrepancyCheck.PT := T#0MS;
   instCmCathodeNgBoxLockUpDown.instTimerDiscrepancyCheck.IN := FALSE;
   instCmCathodeNgBoxLockUpDown.statDisableAlarms := FALSE;
   instCmCathodeNgBoxLockUpDown.statDiagnostics.status := 16#7003;
   instCmCathodeNgBoxLockUpDown.statDiagnostics.subfunctionStatus := 16#0000;
   instCmCathodeNgBoxLockUpDown.statDiagnostics.stateNumber := 0;
   instCmCathodeNgBoxLockUpDown.statEnablePrevious := TRUE;
   instCmCathodeNgBoxLockUpDown.statFirstCall := FALSE;
   instCmCathodeNgBoxLockUpDown.statResetPrevious := FALSE;
   instCmCathodeNgBoxLockUpDown.statValid := TRUE;
   instCmCathodeNgBoxLockUpDown.statBusy := TRUE;
   instCmCathodeNgBoxLockUpDown.statError := FALSE;
   instCmCathodeNgBoxLockUpDown.statInterlockWorkOff := FALSE;
   instCmCathodeNgBoxLockUpDown.statInterlockHomeOff := FALSE;
   instCmCathodeNgBoxLockUpDown.statFbState := 50;
   instCmCathodeNgBoxLockUpDown.statFbStatePrevious := 50;
   instCmCathodeNgBoxLockUpDown.statErrorUserCleared := FALSE;
   instCmCathodeNgBoxLockUpDown.statErrorAutoCleared := FALSE;
   instCmCathodeNgBoxLockUpDown.statErrorState := 16#0000;
   instCmCathodeNgBoxLockUpDown.statDisablingCompleted := FALSE;
   instCmCathodeNgBoxLockUpDown.statFeedbackHomePos := TRUE;
   instCmCathodeNgBoxLockUpDown.statFeedbackWorkPos := FALSE;
   instCmCathodeNgPnpVaccum.enable := TRUE;
   instCmCathodeNgPnpVaccum.parentReferenceDesignator := WSTRING#'';
   instCmCathodeNgPnpVaccum.feedbackHomePos := TRUE;
   instCmCathodeNgPnpVaccum.feedbackWorkPos := FALSE;
   instCmCathodeNgPnpVaccum.enableManualCmds := TRUE;
   instCmCathodeNgPnpVaccum.interlockWorkPos := TRUE;
   instCmCathodeNgPnpVaccum.interlockHomePos := TRUE;
   instCmCathodeNgPnpVaccum.goToHomePos := FALSE;
   instCmCathodeNgPnpVaccum.goToWorkPos := FALSE;
   instCmCathodeNgPnpVaccum.statProcessValues.enable := TRUE;
   instCmCathodeNgPnpVaccum.statProcessValues.referenceDesignator := WSTRING#'NgPnpVaccum';
   instCmCathodeNgPnpVaccum.statProcessValues.commandHomePos := FALSE;
   instCmCathodeNgPnpVaccum.statProcessValues.commandWorkPos := FALSE;
   instCmCathodeNgPnpVaccum.statProcessValues.goToHomePos := FALSE;
   instCmCathodeNgPnpVaccum.statProcessValues.goToWorkPos := FALSE;
   instCmCathodeNgPnpVaccum.statProcessValues.inHomePos := TRUE;
   instCmCathodeNgPnpVaccum.statProcessValues.inWorkPos := FALSE;
   instCmCathodeNgPnpVaccum.statProcessValues.reset := FALSE;
   instCmCathodeNgPnpVaccum.statProcessValues.enableManualCmds := TRUE;
   instCmCathodeNgPnpVaccum.statProcessValues.error := FALSE;
   instCmCathodeNgPnpVaccum.statProcessValues.interlockHomePos := TRUE;
   instCmCathodeNgPnpVaccum.statProcessValues.interlockWorkPos := TRUE;
   instCmCathodeNgPnpVaccum.statProcessValues.status := 16#7003;
   instCmCathodeNgPnpVaccum.statProcessValues.interlockWarningWorkPos := FALSE;
   instCmCathodeNgPnpVaccum.statProcessValues.interlockWarningHomePos := FALSE;
   instCmCathodeNgPnpVaccum.statCurrentInputs.commandHomePos := FALSE;
   instCmCathodeNgPnpVaccum.statCurrentInputs.commandWorkPos := FALSE;
   instCmCathodeNgPnpVaccum.statCurrentInputs.reset := FALSE;
   instCmCathodeNgPnpVaccum.statPreviousInputs.commandHomePos := FALSE;
   instCmCathodeNgPnpVaccum.statPreviousInputs.commandWorkPos := FALSE;
   instCmCathodeNgPnpVaccum.statPreviousInputs.reset := FALSE;
   instCmCathodeNgPnpVaccum.statCurrentInterface.commandHomePos := FALSE;
   instCmCathodeNgPnpVaccum.statCurrentInterface.commandWorkPos := FALSE;
   instCmCathodeNgPnpVaccum.statCurrentInterface.reset := FALSE;
   instCmCathodeNgPnpVaccum.statPreviousInterface.commandHomePos := FALSE;
   instCmCathodeNgPnpVaccum.statPreviousInterface.commandWorkPos := FALSE;
   instCmCathodeNgPnpVaccum.statPreviousInterface.reset := FALSE;
   instCmCathodeNgPnpVaccum.statEmptyDiagnostics.status := 16#0000;
   instCmCathodeNgPnpVaccum.statEmptyDiagnostics.subfunctionStatus := 16#0000;
   instCmCathodeNgPnpVaccum.statEmptyDiagnostics.stateNumber := 0;
   instCmCathodeNgPnpVaccum.instTimerReachPos.PT := T#0MS;
   instCmCathodeNgPnpVaccum.instTimerReachPos.IN := FALSE;
   instCmCathodeNgPnpVaccum.instTimerLeavePos.PT := T#0MS;
   instCmCathodeNgPnpVaccum.instTimerLeavePos.IN := FALSE;
   instCmCathodeNgPnpVaccum.instTimerDiscrepancyCheck.PT := T#0MS;
   instCmCathodeNgPnpVaccum.instTimerDiscrepancyCheck.IN := FALSE;
   instCmCathodeNgPnpVaccum.statDisableAlarms := FALSE;
   instCmCathodeNgPnpVaccum.statDiagnostics.status := 16#7003;
   instCmCathodeNgPnpVaccum.statDiagnostics.subfunctionStatus := 16#0000;
   instCmCathodeNgPnpVaccum.statDiagnostics.stateNumber := 0;
   instCmCathodeNgPnpVaccum.statEnablePrevious := TRUE;
   instCmCathodeNgPnpVaccum.statFirstCall := FALSE;
   instCmCathodeNgPnpVaccum.statResetPrevious := FALSE;
   instCmCathodeNgPnpVaccum.statValid := TRUE;
   instCmCathodeNgPnpVaccum.statBusy := TRUE;
   instCmCathodeNgPnpVaccum.statError := FALSE;
   instCmCathodeNgPnpVaccum.statInterlockWorkOff := FALSE;
   instCmCathodeNgPnpVaccum.statInterlockHomeOff := FALSE;
   instCmCathodeNgPnpVaccum.statFbState := 50;
   instCmCathodeNgPnpVaccum.statFbStatePrevious := 50;
   instCmCathodeNgPnpVaccum.statErrorUserCleared := FALSE;
   instCmCathodeNgPnpVaccum.statErrorAutoCleared := FALSE;
   instCmCathodeNgPnpVaccum.statErrorState := 16#0000;
   instCmCathodeNgPnpVaccum.statDisablingCompleted := FALSE;
   instCmCathodeNgPnpVaccum.statFeedbackHomePos := TRUE;
   instCmCathodeNgPnpVaccum.statFeedbackWorkPos := FALSE;
   instCmCathodeConveyorCoverFwdBwd.enable := TRUE;
   instCmCathodeConveyorCoverFwdBwd.parentReferenceDesignator := WSTRING#'';
   instCmCathodeConveyorCoverFwdBwd.feedbackHomePos := FALSE;
   instCmCathodeConveyorCoverFwdBwd.feedbackWorkPos := FALSE;
   instCmCathodeConveyorCoverFwdBwd.enableManualCmds := TRUE;
   instCmCathodeConveyorCoverFwdBwd.interlockWorkPos := TRUE;
   instCmCathodeConveyorCoverFwdBwd.interlockHomePos := TRUE;
   instCmCathodeConveyorCoverFwdBwd.goToHomePos := FALSE;
   instCmCathodeConveyorCoverFwdBwd.goToWorkPos := FALSE;
   instCmCathodeConveyorCoverFwdBwd.statProcessValues.enable := TRUE;
   instCmCathodeConveyorCoverFwdBwd.statProcessValues.referenceDesignator := WSTRING#'ConveyorCoverFwdBwd';
   instCmCathodeConveyorCoverFwdBwd.statProcessValues.commandHomePos := FALSE;
   instCmCathodeConveyorCoverFwdBwd.statProcessValues.commandWorkPos := FALSE;
   instCmCathodeConveyorCoverFwdBwd.statProcessValues.goToHomePos := FALSE;
   instCmCathodeConveyorCoverFwdBwd.statProcessValues.goToWorkPos := FALSE;
   instCmCathodeConveyorCoverFwdBwd.statProcessValues.inHomePos := FALSE;
   instCmCathodeConveyorCoverFwdBwd.statProcessValues.inWorkPos := FALSE;
   instCmCathodeConveyorCoverFwdBwd.statProcessValues.reset := FALSE;
   instCmCathodeConveyorCoverFwdBwd.statProcessValues.enableManualCmds := TRUE;
   instCmCathodeConveyorCoverFwdBwd.statProcessValues.error := FALSE;
   instCmCathodeConveyorCoverFwdBwd.statProcessValues.interlockHomePos := TRUE;
   instCmCathodeConveyorCoverFwdBwd.statProcessValues.interlockWorkPos := TRUE;
   instCmCathodeConveyorCoverFwdBwd.statProcessValues.status := 16#7003;
   instCmCathodeConveyorCoverFwdBwd.statProcessValues.interlockWarningWorkPos := FALSE;
   instCmCathodeConveyorCoverFwdBwd.statProcessValues.interlockWarningHomePos := FALSE;
   instCmCathodeConveyorCoverFwdBwd.statCurrentInputs.commandHomePos := FALSE;
   instCmCathodeConveyorCoverFwdBwd.statCurrentInputs.commandWorkPos := FALSE;
   instCmCathodeConveyorCoverFwdBwd.statCurrentInputs.reset := FALSE;
   instCmCathodeConveyorCoverFwdBwd.statPreviousInputs.commandHomePos := FALSE;
   instCmCathodeConveyorCoverFwdBwd.statPreviousInputs.commandWorkPos := FALSE;
   instCmCathodeConveyorCoverFwdBwd.statPreviousInputs.reset := FALSE;
   instCmCathodeConveyorCoverFwdBwd.statCurrentInterface.commandHomePos := FALSE;
   instCmCathodeConveyorCoverFwdBwd.statCurrentInterface.commandWorkPos := FALSE;
   instCmCathodeConveyorCoverFwdBwd.statCurrentInterface.reset := FALSE;
   instCmCathodeConveyorCoverFwdBwd.statPreviousInterface.commandHomePos := FALSE;
   instCmCathodeConveyorCoverFwdBwd.statPreviousInterface.commandWorkPos := FALSE;
   instCmCathodeConveyorCoverFwdBwd.statPreviousInterface.reset := FALSE;
   instCmCathodeConveyorCoverFwdBwd.statEmptyDiagnostics.status := 16#0000;
   instCmCathodeConveyorCoverFwdBwd.statEmptyDiagnostics.subfunctionStatus := 16#0000;
   instCmCathodeConveyorCoverFwdBwd.statEmptyDiagnostics.stateNumber := 0;
   instCmCathodeConveyorCoverFwdBwd.instTimerReachPos.PT := T#0MS;
   instCmCathodeConveyorCoverFwdBwd.instTimerReachPos.IN := FALSE;
   instCmCathodeConveyorCoverFwdBwd.instTimerLeavePos.PT := T#0MS;
   instCmCathodeConveyorCoverFwdBwd.instTimerLeavePos.IN := FALSE;
   instCmCathodeConveyorCoverFwdBwd.instTimerDiscrepancyCheck.PT := T#0MS;
   instCmCathodeConveyorCoverFwdBwd.instTimerDiscrepancyCheck.IN := FALSE;
   instCmCathodeConveyorCoverFwdBwd.statDisableAlarms := FALSE;
   instCmCathodeConveyorCoverFwdBwd.statDiagnostics.status := 16#7003;
   instCmCathodeConveyorCoverFwdBwd.statDiagnostics.subfunctionStatus := 16#0000;
   instCmCathodeConveyorCoverFwdBwd.statDiagnostics.stateNumber := 0;
   instCmCathodeConveyorCoverFwdBwd.statEnablePrevious := TRUE;
   instCmCathodeConveyorCoverFwdBwd.statFirstCall := FALSE;
   instCmCathodeConveyorCoverFwdBwd.statResetPrevious := FALSE;
   instCmCathodeConveyorCoverFwdBwd.statValid := TRUE;
   instCmCathodeConveyorCoverFwdBwd.statBusy := TRUE;
   instCmCathodeConveyorCoverFwdBwd.statError := FALSE;
   instCmCathodeConveyorCoverFwdBwd.statInterlockWorkOff := FALSE;
   instCmCathodeConveyorCoverFwdBwd.statInterlockHomeOff := FALSE;
   instCmCathodeConveyorCoverFwdBwd.statFbState := 50;
   instCmCathodeConveyorCoverFwdBwd.statFbStatePrevious := 50;
   instCmCathodeConveyorCoverFwdBwd.statErrorUserCleared := FALSE;
   instCmCathodeConveyorCoverFwdBwd.statErrorAutoCleared := FALSE;
   instCmCathodeConveyorCoverFwdBwd.statErrorState := 16#0000;
   instCmCathodeConveyorCoverFwdBwd.statDisablingCompleted := FALSE;
   instCmCathodeConveyorCoverFwdBwd.statFeedbackHomePos := FALSE;
   instCmCathodeConveyorCoverFwdBwd.statFeedbackWorkPos := FALSE;
   instCmCathodeConveyorPickUpBlower.enable := TRUE;
   instCmCathodeConveyorPickUpBlower.parentReferenceDesignator := WSTRING#'';
   instCmCathodeConveyorPickUpBlower.feedbackHomePos := FALSE;
   instCmCathodeConveyorPickUpBlower.feedbackWorkPos := FALSE;
   instCmCathodeConveyorPickUpBlower.enableManualCmds := TRUE;
   instCmCathodeConveyorPickUpBlower.interlockWorkPos := TRUE;
   instCmCathodeConveyorPickUpBlower.interlockHomePos := TRUE;
   instCmCathodeConveyorPickUpBlower.goToHomePos := FALSE;
   instCmCathodeConveyorPickUpBlower.goToWorkPos := FALSE;
   instCmCathodeConveyorPickUpBlower.statProcessValues.enable := TRUE;
   instCmCathodeConveyorPickUpBlower.statProcessValues.referenceDesignator := WSTRING#'ConveyorPickUpBlower';
   instCmCathodeConveyorPickUpBlower.statProcessValues.commandHomePos := FALSE;
   instCmCathodeConveyorPickUpBlower.statProcessValues.commandWorkPos := FALSE;
   instCmCathodeConveyorPickUpBlower.statProcessValues.goToHomePos := FALSE;
   instCmCathodeConveyorPickUpBlower.statProcessValues.goToWorkPos := FALSE;
   instCmCathodeConveyorPickUpBlower.statProcessValues.inHomePos := FALSE;
   instCmCathodeConveyorPickUpBlower.statProcessValues.inWorkPos := FALSE;
   instCmCathodeConveyorPickUpBlower.statProcessValues.reset := FALSE;
   instCmCathodeConveyorPickUpBlower.statProcessValues.enableManualCmds := TRUE;
   instCmCathodeConveyorPickUpBlower.statProcessValues.error := FALSE;
   instCmCathodeConveyorPickUpBlower.statProcessValues.interlockHomePos := TRUE;
   instCmCathodeConveyorPickUpBlower.statProcessValues.interlockWorkPos := TRUE;
   instCmCathodeConveyorPickUpBlower.statProcessValues.status := 16#7003;
   instCmCathodeConveyorPickUpBlower.statProcessValues.interlockWarningWorkPos := FALSE;
   instCmCathodeConveyorPickUpBlower.statProcessValues.interlockWarningHomePos := FALSE;
   instCmCathodeConveyorPickUpBlower.statCurrentInputs.commandHomePos := FALSE;
   instCmCathodeConveyorPickUpBlower.statCurrentInputs.commandWorkPos := FALSE;
   instCmCathodeConveyorPickUpBlower.statCurrentInputs.reset := FALSE;
   instCmCathodeConveyorPickUpBlower.statPreviousInputs.commandHomePos := FALSE;
   instCmCathodeConveyorPickUpBlower.statPreviousInputs.commandWorkPos := FALSE;
   instCmCathodeConveyorPickUpBlower.statPreviousInputs.reset := FALSE;
   instCmCathodeConveyorPickUpBlower.statCurrentInterface.commandHomePos := FALSE;
   instCmCathodeConveyorPickUpBlower.statCurrentInterface.commandWorkPos := FALSE;
   instCmCathodeConveyorPickUpBlower.statCurrentInterface.reset := FALSE;
   instCmCathodeConveyorPickUpBlower.statPreviousInterface.commandHomePos := FALSE;
   instCmCathodeConveyorPickUpBlower.statPreviousInterface.commandWorkPos := FALSE;
   instCmCathodeConveyorPickUpBlower.statPreviousInterface.reset := FALSE;
   instCmCathodeConveyorPickUpBlower.statEmptyDiagnostics.status := 16#0000;
   instCmCathodeConveyorPickUpBlower.statEmptyDiagnostics.subfunctionStatus := 16#0000;
   instCmCathodeConveyorPickUpBlower.statEmptyDiagnostics.stateNumber := 0;
   instCmCathodeConveyorPickUpBlower.instTimerReachPos.PT := T#0MS;
   instCmCathodeConveyorPickUpBlower.instTimerReachPos.IN := FALSE;
   instCmCathodeConveyorPickUpBlower.instTimerLeavePos.PT := T#0MS;
   instCmCathodeConveyorPickUpBlower.instTimerLeavePos.IN := FALSE;
   instCmCathodeConveyorPickUpBlower.instTimerDiscrepancyCheck.PT := T#0MS;
   instCmCathodeConveyorPickUpBlower.instTimerDiscrepancyCheck.IN := FALSE;
   instCmCathodeConveyorPickUpBlower.statDisableAlarms := FALSE;
   instCmCathodeConveyorPickUpBlower.statDiagnostics.status := 16#7003;
   instCmCathodeConveyorPickUpBlower.statDiagnostics.subfunctionStatus := 16#0000;
   instCmCathodeConveyorPickUpBlower.statDiagnostics.stateNumber := 0;
   instCmCathodeConveyorPickUpBlower.statEnablePrevious := TRUE;
   instCmCathodeConveyorPickUpBlower.statFirstCall := FALSE;
   instCmCathodeConveyorPickUpBlower.statResetPrevious := FALSE;
   instCmCathodeConveyorPickUpBlower.statValid := TRUE;
   instCmCathodeConveyorPickUpBlower.statBusy := TRUE;
   instCmCathodeConveyorPickUpBlower.statError := FALSE;
   instCmCathodeConveyorPickUpBlower.statInterlockWorkOff := FALSE;
   instCmCathodeConveyorPickUpBlower.statInterlockHomeOff := FALSE;
   instCmCathodeConveyorPickUpBlower.statFbState := 50;
   instCmCathodeConveyorPickUpBlower.statFbStatePrevious := 50;
   instCmCathodeConveyorPickUpBlower.statErrorUserCleared := FALSE;
   instCmCathodeConveyorPickUpBlower.statErrorAutoCleared := FALSE;
   instCmCathodeConveyorPickUpBlower.statErrorState := 16#0000;
   instCmCathodeConveyorPickUpBlower.statDisablingCompleted := FALSE;
   instCmCathodeConveyorPickUpBlower.statFeedbackHomePos := FALSE;
   instCmCathodeConveyorPickUpBlower.statFeedbackWorkPos := FALSE;
   instManageAlarms.proDiagState.Total_Number := 497;
   instManageAlarms.proDiagState.All := TRUE;
   instManageAlarms.proDiagState.O := FALSE;
   instManageAlarms.proDiagState.I := FALSE;
   instManageAlarms.proDiagState.R := FALSE;
   instManageAlarms.proDiagState."A" := FALSE;
   instManageAlarms.proDiagState.P := FALSE;
   instManageAlarms.proDiagState.Merr := TRUE;
   instManageAlarms.proDiagState.Mtxt := FALSE;
   instManageAlarms.proDiagState.SV_Types := 16#20;
   instManageAlarms.proDiagState.C1 := TRUE;
   instManageAlarms.proDiagState.C2 := FALSE;
   instManageAlarms.proDiagState.C3 := FALSE;
   instManageAlarms.proDiagState.C4 := FALSE;
   instManageAlarms.proDiagState.C5 := FALSE;
   instManageAlarms.proDiagState.C6 := FALSE;
   instManageAlarms.proDiagState.C7 := FALSE;
   instManageAlarms.proDiagState.C8 := FALSE;
   instManageAlarms.proDiagState.Categories := 16#01;
   instManageAlarms.proDiagState.Sub_Cat_1 := 16#0000_0001;
   instManageAlarms.proDiagState.Sub_Cat_2 := 16#0000_0000;
   instManageAlarms.proDiagState.Reserved := 16#00;
   instManageAlarms.parentAlarmDB.error := TRUE;
   instManageAlarms.parentAlarmDB.warning := FALSE;
   instManageAlarms.parentAlarmDB.info := FALSE;
   instManageAlarms.alarmDB.error := TRUE;
   instManageAlarms.alarmDB.warning := FALSE;
   instManageAlarms.alarmDB.info := FALSE;
   instManageAlarms.hmiInterfaceDB.error := TRUE;
   instManageAlarms.hmiInterfaceDB.warning := FALSE;
   instManageAlarms.hmiInterfaceDB.info := FALSE;
   statUnitStatus.acknowledgeActive := FALSE;
   statUnitStatus.alarmsDisabled := FALSE;
   statUnitStatus.simulationActive := FALSE;
   statUnitStatus.safetyReleased := TRUE;
   statUnitStatus.state.current := 2;
   statUnitStatus.state.clearing := FALSE;
   statUnitStatus.state.stopped := TRUE;
   statUnitStatus.state.starting := FALSE;
   statUnitStatus.state.idle := FALSE;
   statUnitStatus.state.suspended := FALSE;
   statUnitStatus.state.execute := FALSE;
   statUnitStatus.state.stopping := FALSE;
   statUnitStatus.state.aborting := FALSE;
   statUnitStatus.state.aborted := FALSE;
   statUnitStatus.state.holding := FALSE;
   statUnitStatus.state.held := FALSE;
   statUnitStatus.state.unholding := FALSE;
   statUnitStatus.state.suspending := FALSE;
   statUnitStatus.state.unsuspending := FALSE;
   statUnitStatus.state.resetting := FALSE;
   statUnitStatus.state.completing := FALSE;
   statUnitStatus.state.complete := FALSE;
END_DATA_BLOCK
